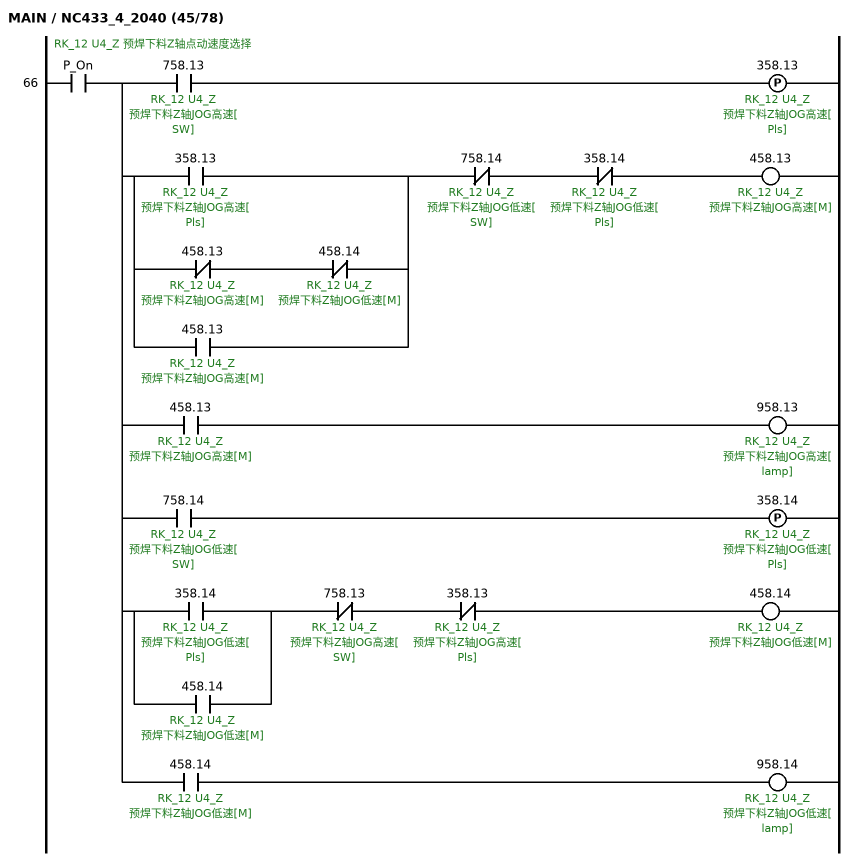
; [picture p192: MAIN / NC433_4_2040, rungs 66-66]
; rung 66: RK_12 U4_Z 预焊下料Z轴点动速度选择
LD P_On
OUT TR0
AND 758.13  ; RK_12 U4_Z 预焊下料Z轴JOG高速[SW]
DIFU(013) 358.13  ; RK_12 U4_Z 预焊下料Z轴JOG高速[Pls]
LD TR0
LD 358.13  ; RK_12 U4_Z 预焊下料Z轴JOG高速[Pls]
LDNOT 458.13  ; RK_12 U4_Z 预焊下料Z轴JOG高速[M]
ANDNOT 458.14  ; RK_12 U4_Z 预焊下料Z轴JOG低速[M]
ORLD
OR 458.13  ; RK_12 U4_Z 预焊下料Z轴JOG高速[M]
ANDLD
ANDNOT 758.14  ; RK_12 U4_Z 预焊下料Z轴JOG低速[SW]
ANDNOT 358.14  ; RK_12 U4_Z 预焊下料Z轴JOG低速[Pls]
OUT 458.13  ; RK_12 U4_Z 预焊下料Z轴JOG高速[M]
LD TR0
AND 458.13  ; RK_12 U4_Z 预焊下料Z轴JOG高速[M]
OUT 958.13  ; RK_12 U4_Z 预焊下料Z轴JOG高速[lamp]
LD TR0
AND 758.14  ; RK_12 U4_Z 预焊下料Z轴JOG低速[SW]
DIFU(013) 358.14  ; RK_12 U4_Z 预焊下料Z轴JOG低速[Pls]
LD TR0
LD 358.14  ; RK_12 U4_Z 预焊下料Z轴JOG低速[Pls]
OR 458.14  ; RK_12 U4_Z 预焊下料Z轴JOG低速[M]
ANDLD
ANDNOT 758.13  ; RK_12 U4_Z 预焊下料Z轴JOG高速[SW]
ANDNOT 358.13  ; RK_12 U4_Z 预焊下料Z轴JOG高速[Pls]
OUT 458.14  ; RK_12 U4_Z 预焊下料Z轴JOG低速[M]
LD TR0
AND 458.14  ; RK_12 U4_Z 预焊下料Z轴JOG低速[M]
OUT 958.14  ; RK_12 U4_Z 预焊下料Z轴JOG低速[lamp]

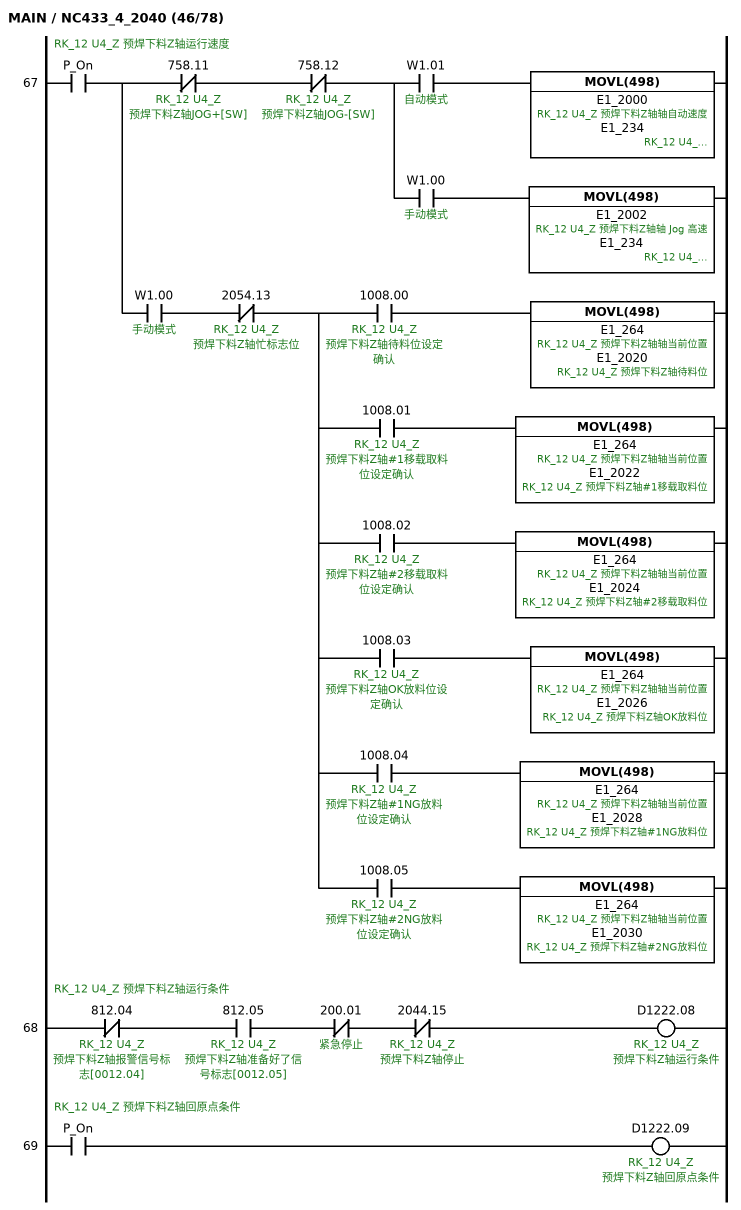
; rung 67: RK_12 U4_Z 预焊下料Z轴运行速度
LD P_On
OUT TR0
ANDNOT 758.11  ; RK_12 U4_Z 预焊下料Z轴JOG+[SW]
ANDNOT 758.12  ; RK_12 U4_Z 预焊下料Z轴JOG-[SW]
OUT TR1
AND W1.01  ; 自动模式
MOVL(498) E1_2000 E1_234  ; RK_12 U4_Z 预焊下料Z轴轴自动速度, RK_12 U4_Z 预焊下料Z轴轴直接操作速度
LD TR1
AND W1.00  ; 手动模式
MOVL(498) E1_2002 E1_234  ; RK_12 U4_Z 预焊下料Z轴轴 Jog 高速, RK_12 U4_Z 预焊下料Z轴轴直接操作速度
LD TR0
AND W1.00  ; 手动模式
ANDNOT 2054.13  ; RK_12 U4_Z 预焊下料Z轴忙标志位
OUT TR0
AND 1008.00  ; RK_12 U4_Z 预焊下料Z轴待料位设定确认
MOVL(498) E1_264 E1_2020  ; RK_12 U4_Z 预焊下料Z轴轴当前位置, RK_12 U4_Z 预焊下料Z轴待料位
LD TR0
AND 1008.01  ; RK_12 U4_Z 预焊下料Z轴#1移载取料位设定确认
MOVL(498) E1_264 E1_2022  ; RK_12 U4_Z 预焊下料Z轴轴当前位置, RK_12 U4_Z 预焊下料Z轴#1移载取料位
LD TR0
AND 1008.02  ; RK_12 U4_Z 预焊下料Z轴#2移载取料位设定确认
MOVL(498) E1_264 E1_2024  ; RK_12 U4_Z 预焊下料Z轴轴当前位置, RK_12 U4_Z 预焊下料Z轴#2移载取料位
LD TR0
AND 1008.03  ; RK_12 U4_Z 预焊下料Z轴OK放料位设定确认
MOVL(498) E1_264 E1_2026  ; RK_12 U4_Z 预焊下料Z轴轴当前位置, RK_12 U4_Z 预焊下料Z轴OK放料位
LD TR0
AND 1008.04  ; RK_12 U4_Z 预焊下料Z轴#1NG放料位设定确认
MOVL(498) E1_264 E1_2028  ; RK_12 U4_Z 预焊下料Z轴轴当前位置, RK_12 U4_Z 预焊下料Z轴#1NG放料位
LD TR0
AND 1008.05  ; RK_12 U4_Z 预焊下料Z轴#2NG放料位设定确认
MOVL(498) E1_264 E1_2030  ; RK_12 U4_Z 预焊下料Z轴轴当前位置, RK_12 U4_Z 预焊下料Z轴#2NG放料位
; rung 68: RK_12 U4_Z 预焊下料Z轴运行条件
LDNOT 812.04  ; RK_12 U4_Z 预焊下料Z轴报警信号标志[0012.04]
AND 812.05  ; RK_12 U4_Z 预焊下料Z轴准备好了信号标志[0012.05]
ANDNOT 200.01  ; 紧急停止
ANDNOT 2044.15  ; RK_12 U4_Z 预焊下料Z轴停止
OUT D1222.08  ; RK_12 U4_Z 预焊下料Z轴运行条件
; rung 69: RK_12 U4_Z 预焊下料Z轴回原点条件
LD P_On
OUT D1222.09  ; RK_12 U4_Z 预焊下料Z轴回原点条件

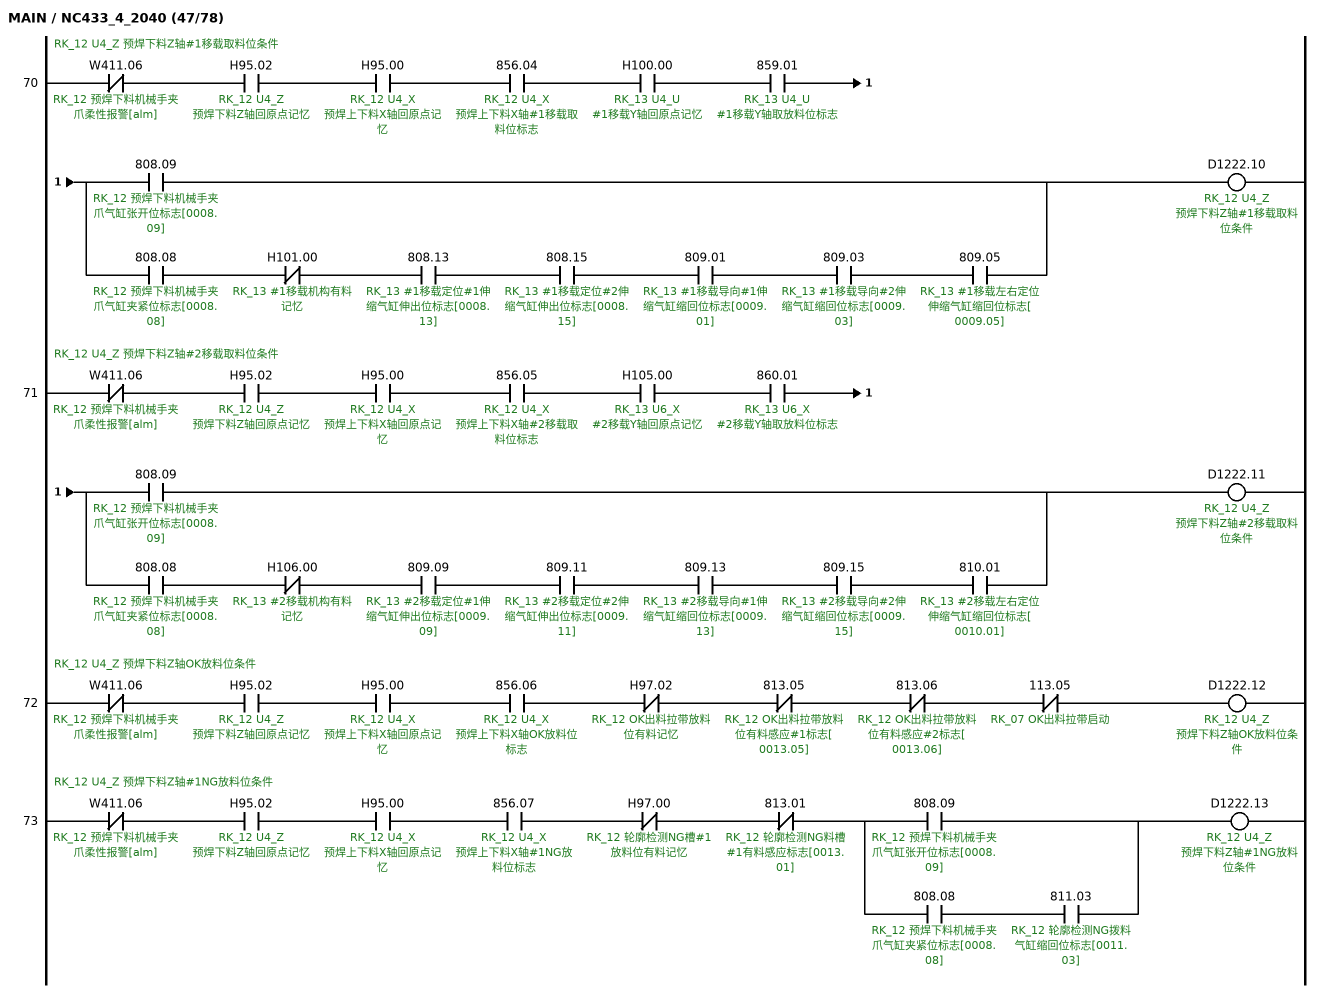
; rung 70: RK_12 U4_Z 预焊下料Z轴#1移载取料位条件
LDNOT W411.06  ; RK_12 预焊下料机械手夹爪柔性报警[alm]
AND H95.02  ; RK_12 U4_Z 预焊下料Z轴回原点记忆
AND H95.00  ; RK_12 U4_X 预焊上下料X轴回原点记忆
AND 856.04  ; RK_12 U4_X 预焊上下料X轴#1移载取料位标志
AND H100.00  ; RK_13 U4_U #1移载Y轴回原点记忆
AND 859.01  ; RK_13 U4_U #1移载Y轴取放料位标志
LD 808.09  ; RK_12 预焊下料机械手夹爪气缸张开位标志[0008.09]
LD 808.08  ; RK_12 预焊下料机械手夹爪气缸夹紧位标志[0008.08]
ANDNOT H101.00  ; RK_13 #1移载机构有料记忆
AND 808.13  ; RK_13 #1移载定位#1伸缩气缸伸出位标志[0008.13]
AND 808.15  ; RK_13 #1移载定位#2伸缩气缸伸出位标志[0008.15]
AND 809.01  ; RK_13 #1移载导向#1伸缩气缸缩回位标志[0009.01]
AND 809.03  ; RK_13 #1移载导向#2伸缩气缸缩回位标志[0009.03]
AND 809.05  ; RK_13 #1移载左右定位伸缩气缸缩回位标志[0009.05]
ORLD
ANDLD
OUT D1222.10  ; RK_12 U4_Z 预焊下料Z轴#1移载取料位条件
; rung 71: RK_12 U4_Z 预焊下料Z轴#2移载取料位条件
LDNOT W411.06  ; RK_12 预焊下料机械手夹爪柔性报警[alm]
AND H95.02  ; RK_12 U4_Z 预焊下料Z轴回原点记忆
AND H95.00  ; RK_12 U4_X 预焊上下料X轴回原点记忆
AND 856.05  ; RK_12 U4_X 预焊上下料X轴#2移载取料位标志
AND H105.00  ; RK_13 U6_X #2移载Y轴回原点记忆
AND 860.01  ; RK_13 U6_X #2移载Y轴取放料位标志
LD 808.09  ; RK_12 预焊下料机械手夹爪气缸张开位标志[0008.09]
LD 808.08  ; RK_12 预焊下料机械手夹爪气缸夹紧位标志[0008.08]
ANDNOT H106.00  ; RK_13 #2移载机构有料记忆
AND 809.09  ; RK_13 #2移载定位#1伸缩气缸伸出位标志[0009.09]
AND 809.11  ; RK_13 #2移载定位#2伸缩气缸伸出位标志[0009.11]
AND 809.13  ; RK_13 #2移载导向#1伸缩气缸缩回位标志[0009.13]
AND 809.15  ; RK_13 #2移载导向#2伸缩气缸缩回位标志[0009.15]
AND 810.01  ; RK_13 #2移载左右定位伸缩气缸缩回位标志[0010.01]
ORLD
ANDLD
OUT D1222.11  ; RK_12 U4_Z 预焊下料Z轴#2移载取料位条件
; rung 72: RK_12 U4_Z 预焊下料Z轴OK放料位条件
LDNOT W411.06  ; RK_12 预焊下料机械手夹爪柔性报警[alm]
AND H95.02  ; RK_12 U4_Z 预焊下料Z轴回原点记忆
AND H95.00  ; RK_12 U4_X 预焊上下料X轴回原点记忆
AND 856.06  ; RK_12 U4_X 预焊上下料X轴OK放料位标志
ANDNOT H97.02  ; RK_12 OK出料拉带放料位有料记忆  // RK_12 OK出料拉带放料位有料记忆+OK出料拉带放料位有料感应标志+拉带电机未启动标志！！
ANDNOT 813.05  ; RK_12 OK出料拉带放料位有料感应#1标志[0013.05]
ANDNOT 813.06  ; RK_12 OK出料拉带放料位有料感应#2标志[0013.06]
ANDNOT 113.05  ; RK_07 OK出料拉带启动
OUT D1222.12  ; RK_12 U4_Z 预焊下料Z轴OK放料位条件
; rung 73: RK_12 U4_Z 预焊下料Z轴#1NG放料位条件
LDNOT W411.06  ; RK_12 预焊下料机械手夹爪柔性报警[alm]
AND H95.02  ; RK_12 U4_Z 预焊下料Z轴回原点记忆
AND H95.00  ; RK_12 U4_X 预焊上下料X轴回原点记忆
AND 856.07  ; RK_12 U4_X 预焊上下料X轴#1NG放料位标志
ANDNOT H97.00  ; RK_12 轮廓检测NG槽#1放料位有料记忆
ANDNOT 813.01  ; RK_12 轮廓检测NG料槽#1有料感应标志[0013.01]
LD 808.09  ; RK_12 预焊下料机械手夹爪气缸张开位标志[0008.09]
LD 808.08  ; RK_12 预焊下料机械手夹爪气缸夹紧位标志[0008.08]
AND 811.03  ; RK_12 轮廓检测NG拨料气缸缩回位标志[0011.03]
ORLD
ANDLD
OUT D1222.13  ; RK_12 U4_Z 预焊下料Z轴#1NG放料位条件

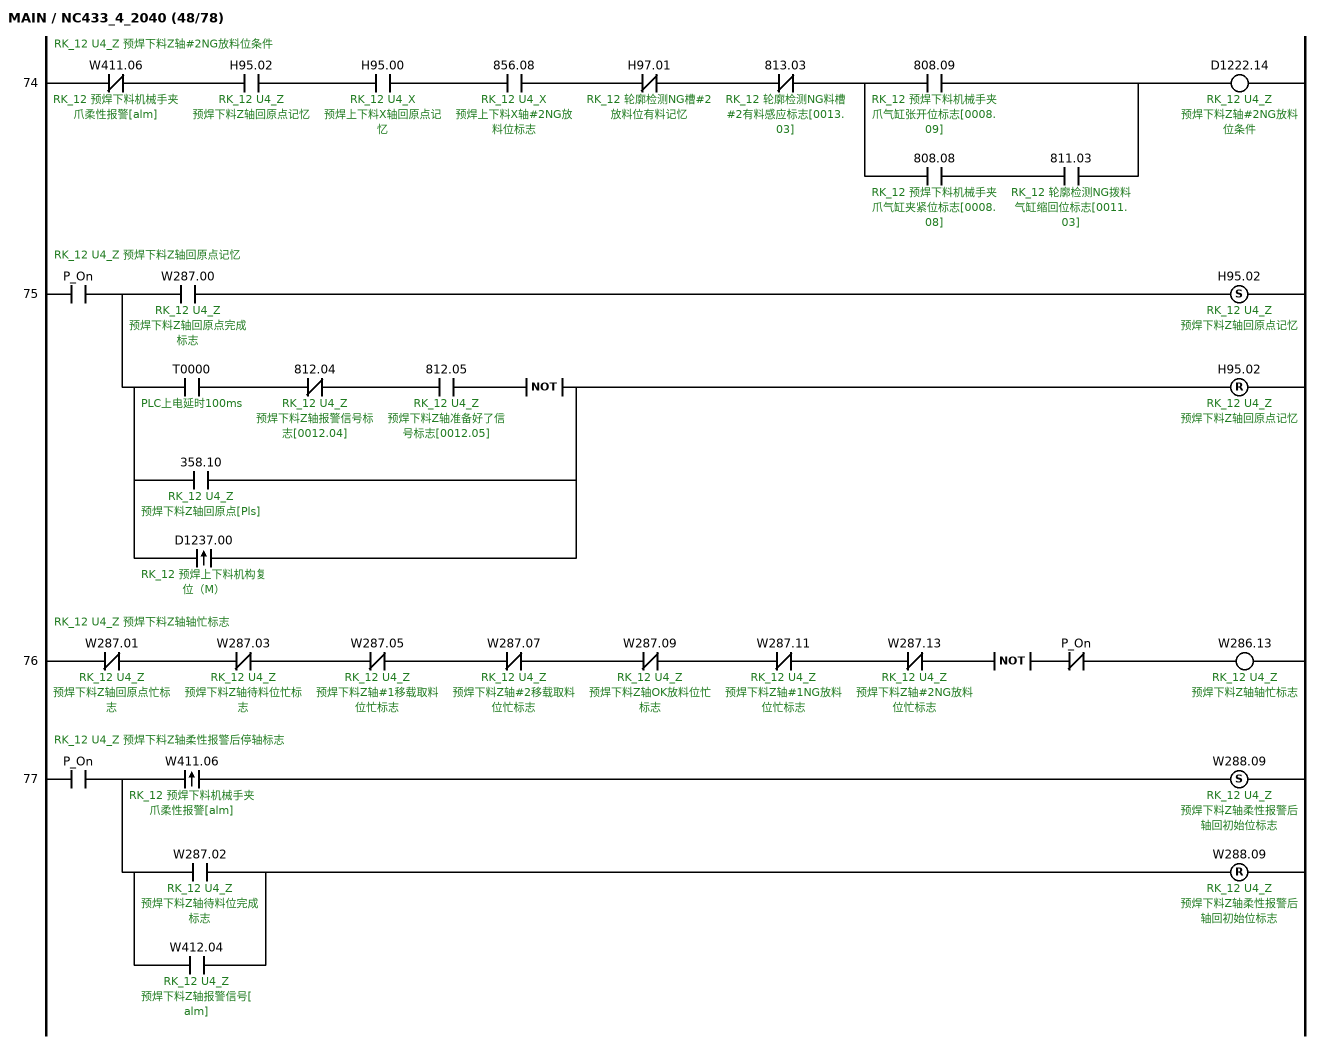
; rung 74: RK_12 U4_Z 预焊下料Z轴#2NG放料位条件
LDNOT W411.06  ; RK_12 预焊下料机械手夹爪柔性报警[alm]
AND H95.02  ; RK_12 U4_Z 预焊下料Z轴回原点记忆
AND H95.00  ; RK_12 U4_X 预焊上下料X轴回原点记忆
AND 856.08  ; RK_12 U4_X 预焊上下料X轴#2NG放料位标志
ANDNOT H97.01  ; RK_12 轮廓检测NG槽#2放料位有料记忆
ANDNOT 813.03  ; RK_12 轮廓检测NG料槽#2有料感应标志[0013.03]
LD 808.09  ; RK_12 预焊下料机械手夹爪气缸张开位标志[0008.09]
LD 808.08  ; RK_12 预焊下料机械手夹爪气缸夹紧位标志[0008.08]
AND 811.03  ; RK_12 轮廓检测NG拨料气缸缩回位标志[0011.03]
ORLD
ANDLD
OUT D1222.14  ; RK_12 U4_Z 预焊下料Z轴#2NG放料位条件
; rung 75: RK_12 U4_Z 预焊下料Z轴回原点记忆
LD P_On
OUT TR0
AND W287.00  ; RK_12 U4_Z 预焊下料Z轴回原点完成标志
SET H95.02  ; RK_12 U4_Z 预焊下料Z轴回原点记忆
LD TR0
LD T0000  ; PLC上电延时100ms
ANDNOT 812.04  ; RK_12 U4_Z 预焊下料Z轴报警信号标志[0012.04]
AND 812.05  ; RK_12 U4_Z 预焊下料Z轴准备好了信号标志[0012.05]
NOT(520)
OR 358.10  ; RK_12 U4_Z 预焊下料Z轴回原点[Pls]
@OR D1237.00  ; RK_12 预焊上下料机构复位（M）
ANDLD
RSET H95.02  ; RK_12 U4_Z 预焊下料Z轴回原点记忆
; rung 76: RK_12 U4_Z 预焊下料Z轴轴忙标志
LDNOT W287.01  ; RK_12 U4_Z 预焊下料Z轴回原点忙标志
ANDNOT W287.03  ; RK_12 U4_Z 预焊下料Z轴待料位忙标志
ANDNOT W287.05  ; RK_12 U4_Z 预焊下料Z轴#1移载取料位忙标志
ANDNOT W287.07  ; RK_12 U4_Z 预焊下料Z轴#2移载取料位忙标志
ANDNOT W287.09  ; RK_12 U4_Z 预焊下料Z轴OK放料位忙标志
ANDNOT W287.11  ; RK_12 U4_Z 预焊下料Z轴#1NG放料位忙标志
ANDNOT W287.13  ; RK_12 U4_Z 预焊下料Z轴#2NG放料位忙标志
NOT(520)
ANDNOT P_On
OUT W286.13  ; RK_12 U4_Z 预焊下料Z轴轴忙标志
; rung 77: RK_12 U4_Z 预焊下料Z轴柔性报警后停轴标志
LD P_On
OUT TR0
@AND W411.06  ; RK_12 预焊下料机械手夹爪柔性报警[alm]
SET W288.09  ; RK_12 U4_Z 预焊下料Z轴柔性报警后轴回初始位标志
LD TR0
LD W287.02  ; RK_12 U4_Z 预焊下料Z轴待料位完成标志
OR W412.04  ; RK_12 U4_Z 预焊下料Z轴报警信号[alm]
ANDLD
RSET W288.09  ; RK_12 U4_Z 预焊下料Z轴柔性报警后轴回初始位标志

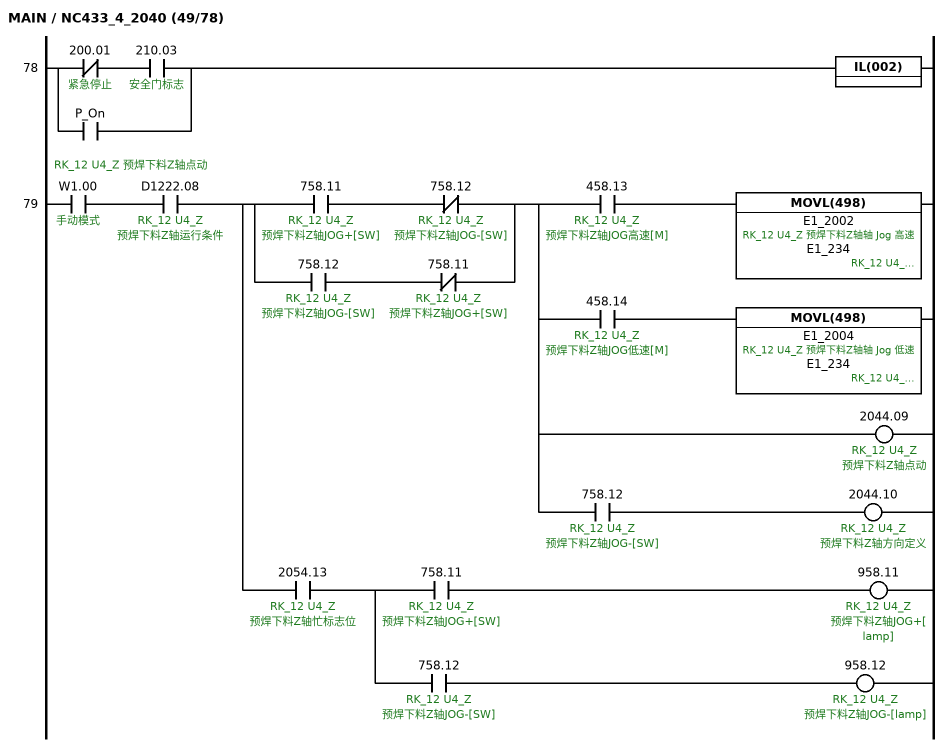
; rung 78
LDNOT 200.01  ; 紧急停止
AND 210.03  ; 安全门标志
OR P_On
IL(002)
; rung 79: RK_12 U4_Z 预焊下料Z轴点动
LD W1.00  ; 手动模式
AND D1222.08  ; RK_12 U4_Z 预焊下料Z轴运行条件
OUT TR0
LD 758.11  ; RK_12 U4_Z 预焊下料Z轴JOG+[SW]
ANDNOT 758.12  ; RK_12 U4_Z 预焊下料Z轴JOG-[SW]
LD 758.12  ; RK_12 U4_Z 预焊下料Z轴JOG-[SW]
ANDNOT 758.11  ; RK_12 U4_Z 预焊下料Z轴JOG+[SW]
ORLD
ANDLD
OUT TR1
AND 458.13  ; RK_12 U4_Z 预焊下料Z轴JOG高速[M]
MOVL(498) E1_2002 E1_234  ; RK_12 U4_Z 预焊下料Z轴轴 Jog 高速, RK_12 U4_Z 预焊下料Z轴轴直接操作速度
LD TR1
AND 458.14  ; RK_12 U4_Z 预焊下料Z轴JOG低速[M]
MOVL(498) E1_2004 E1_234  ; RK_12 U4_Z 预焊下料Z轴轴 Jog 低速, RK_12 U4_Z 预焊下料Z轴轴直接操作速度
LD TR1
OUT 2044.09  ; RK_12 U4_Z 预焊下料Z轴点动
AND 758.12  ; RK_12 U4_Z 预焊下料Z轴JOG-[SW]
OUT 2044.10  ; RK_12 U4_Z 预焊下料Z轴方向定义
LD TR0
AND 2054.13  ; RK_12 U4_Z 预焊下料Z轴忙标志位
OUT TR0
AND 758.11  ; RK_12 U4_Z 预焊下料Z轴JOG+[SW]
OUT 958.11  ; RK_12 U4_Z 预焊下料Z轴JOG+[lamp]
LD TR0
AND 758.12  ; RK_12 U4_Z 预焊下料Z轴JOG-[SW]
OUT 958.12  ; RK_12 U4_Z 预焊下料Z轴JOG-[lamp]

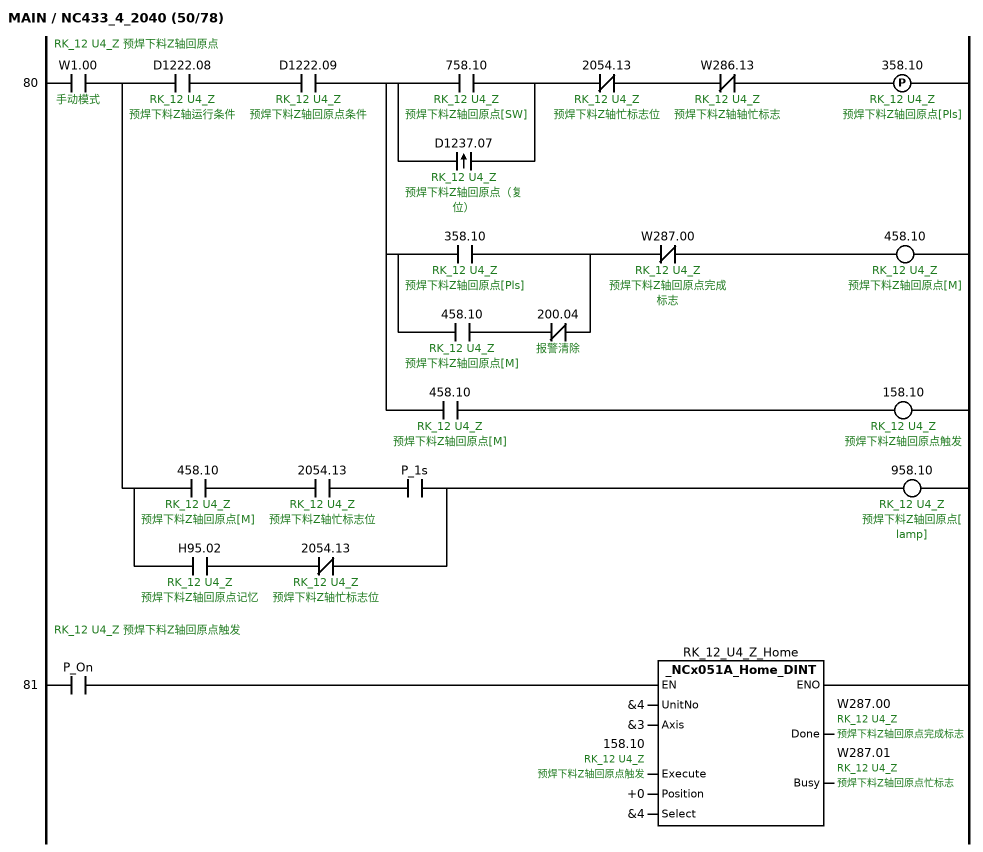
; rung 80: RK_12 U4_Z 预焊下料Z轴回原点
LD W1.00  ; 手动模式
OUT TR0
AND D1222.08  ; RK_12 U4_Z 预焊下料Z轴运行条件
AND D1222.09  ; RK_12 U4_Z 预焊下料Z轴回原点条件
OUT TR1
LD 758.10  ; RK_12 U4_Z 预焊下料Z轴回原点[SW]
@OR D1237.07  ; RK_12 U4_Z 预焊下料Z轴回原点（复位）
ANDLD
ANDNOT 2054.13  ; RK_12 U4_Z 预焊下料Z轴忙标志位
ANDNOT W286.13  ; RK_12 U4_Z 预焊下料Z轴轴忙标志
DIFU(013) 358.10  ; RK_12 U4_Z 预焊下料Z轴回原点[Pls]
LD TR1
LD 358.10  ; RK_12 U4_Z 预焊下料Z轴回原点[Pls]
LD 458.10  ; RK_12 U4_Z 预焊下料Z轴回原点[M]
ANDNOT 200.04  ; 报警清除
ORLD
ANDLD
ANDNOT W287.00  ; RK_12 U4_Z 预焊下料Z轴回原点完成标志
OUT 458.10  ; RK_12 U4_Z 预焊下料Z轴回原点[M]
LD TR1
AND 458.10  ; RK_12 U4_Z 预焊下料Z轴回原点[M]
OUT 158.10  ; RK_12 U4_Z 预焊下料Z轴回原点触发
LD TR0
LD 458.10  ; RK_12 U4_Z 预焊下料Z轴回原点[M]
AND 2054.13  ; RK_12 U4_Z 预焊下料Z轴忙标志位
AND P_1s
LD H95.02  ; RK_12 U4_Z 预焊下料Z轴回原点记忆
ANDNOT 2054.13  ; RK_12 U4_Z 预焊下料Z轴忙标志位
ORLD
ANDLD
OUT 958.10  ; RK_12 U4_Z 预焊下料Z轴回原点[lamp]
; rung 81: RK_12 U4_Z 预焊下料Z轴回原点触发
LD P_On
CALL RK_12_U4_Z_Home : _NCx051A_Home_DINT (UnitNo := &4, Axis := &3, Execute := 158.10, Position := +0, Select := &4, Done => W287.00, Busy => W287.01)  ; RK_12 U4_Z 预焊下料Z轴回原点触发, RK_12 U4_Z 预焊下料Z轴回原点完成标志, RK_12 U4_Z 预焊下料Z轴回原点忙标志

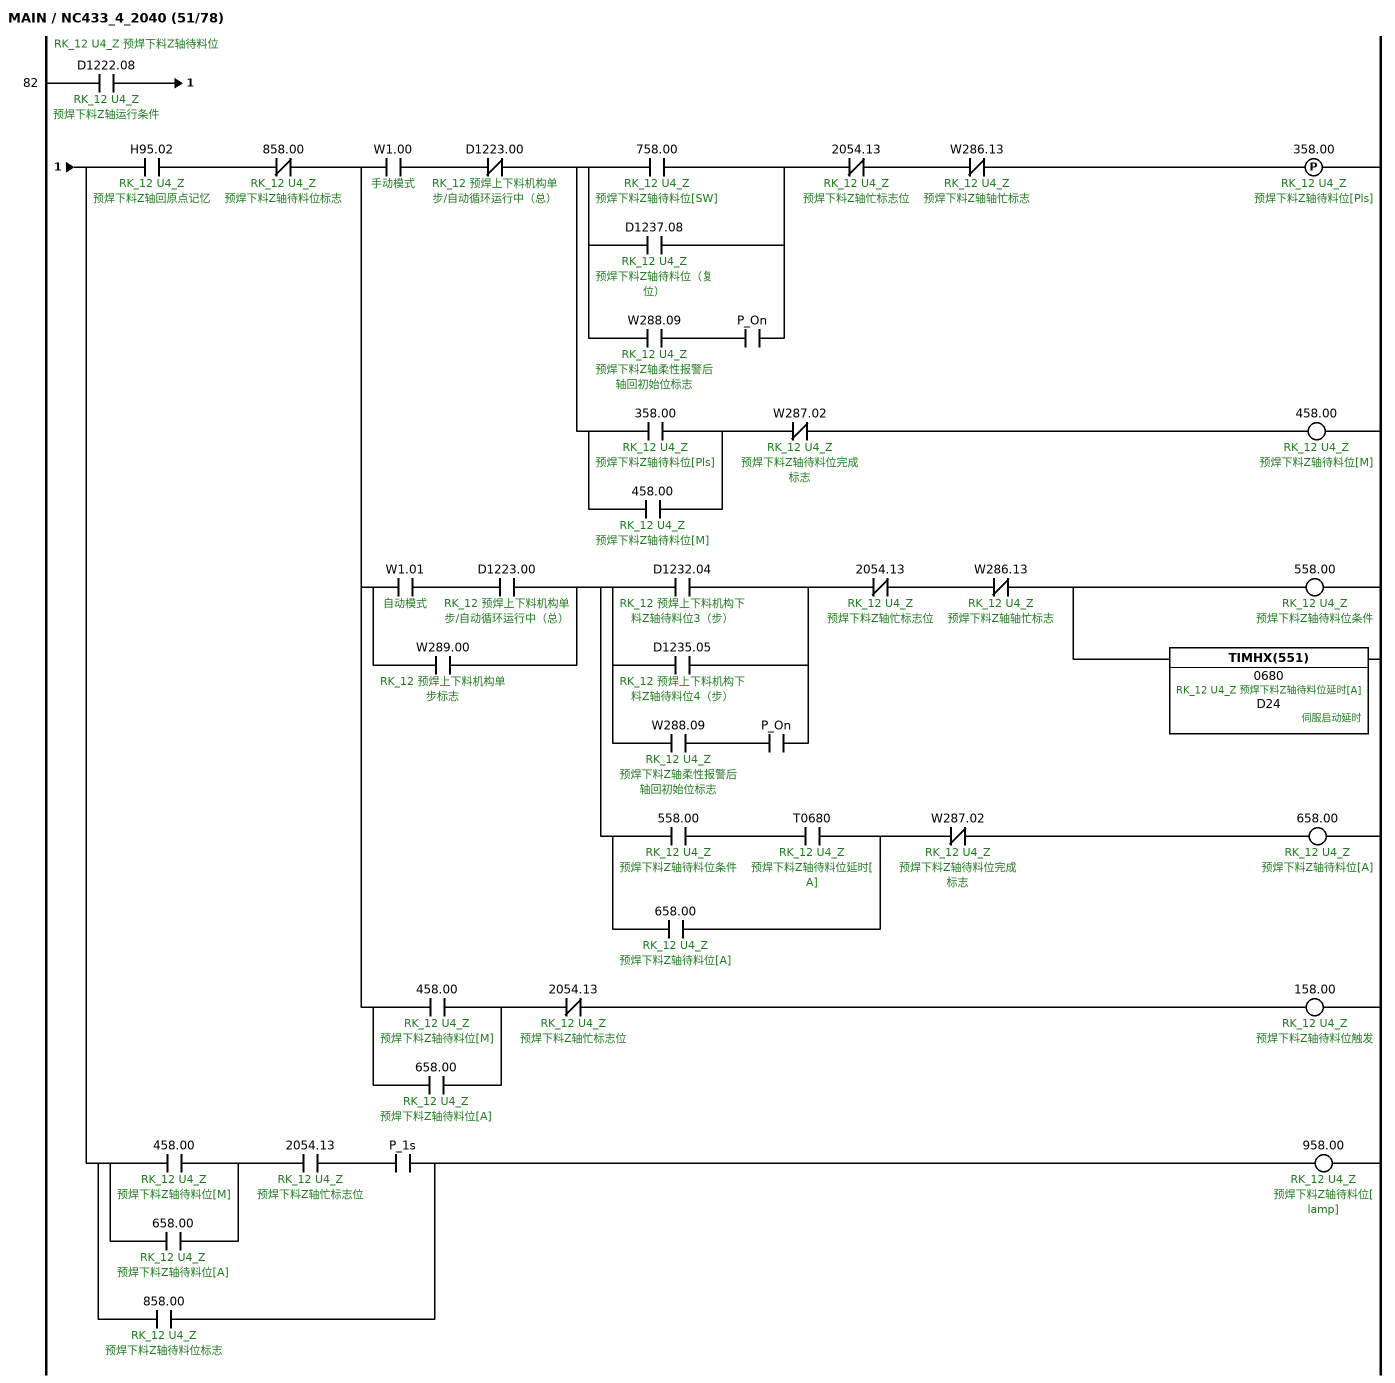
; rung 82: RK_12 U4_Z 预焊下料Z轴待料位
LD D1222.08  ; RK_12 U4_Z 预焊下料Z轴运行条件
OUT TR0
AND H95.02  ; RK_12 U4_Z 预焊下料Z轴回原点记忆
ANDNOT 858.00  ; RK_12 U4_Z 预焊下料Z轴待料位标志
OUT TR1
AND W1.00  ; 手动模式
ANDNOT D1223.00  ; RK_12 预焊上下料机构单步/自动循环运行中（总）
OUT TR2
LD 758.00  ; RK_12 U4_Z 预焊下料Z轴待料位[SW]
OR D1237.08  ; RK_12 U4_Z 预焊下料Z轴待料位（复位）
LD W288.09  ; RK_12 U4_Z 预焊下料Z轴柔性报警后轴回初始位标志
AND P_On
ORLD
ANDLD
ANDNOT 2054.13  ; RK_12 U4_Z 预焊下料Z轴忙标志位
ANDNOT W286.13  ; RK_12 U4_Z 预焊下料Z轴轴忙标志
DIFU(013) 358.00  ; RK_12 U4_Z 预焊下料Z轴待料位[Pls]
LD TR2
LD 358.00  ; RK_12 U4_Z 预焊下料Z轴待料位[Pls]
OR 458.00  ; RK_12 U4_Z 预焊下料Z轴待料位[M]
ANDLD
ANDNOT W287.02  ; RK_12 U4_Z 预焊下料Z轴待料位完成标志
OUT 458.00  ; RK_12 U4_Z 预焊下料Z轴待料位[M]
LD TR1
LD W1.01  ; 自动模式
AND D1223.00  ; RK_12 预焊上下料机构单步/自动循环运行中（总）
OR W289.00  ; RK_12 预焊上下料机构单步标志
ANDLD
OUT TR2
LD D1232.04  ; RK_12 预焊上下料机构下料Z轴待料位3（步）
OR D1235.05  ; RK_12 预焊上下料机构下料Z轴待料位4（步）
LD W288.09  ; RK_12 U4_Z 预焊下料Z轴柔性报警后轴回初始位标志
AND P_On
ORLD
ANDLD
ANDNOT 2054.13  ; RK_12 U4_Z 预焊下料Z轴忙标志位
ANDNOT W286.13  ; RK_12 U4_Z 预焊下料Z轴轴忙标志
OUT 558.00  ; RK_12 U4_Z 预焊下料Z轴待料位条件
TIMHX(551) 0680 D24  ; 伺服启动延时, RK_12 U4_Z 预焊下料Z轴待料位延时[A]
LD TR2
LD 558.00  ; RK_12 U4_Z 预焊下料Z轴待料位条件
AND T0680  ; RK_12 U4_Z 预焊下料Z轴待料位延时[A]
OR 658.00  ; RK_12 U4_Z 预焊下料Z轴待料位[A]
ANDLD
ANDNOT W287.02  ; RK_12 U4_Z 预焊下料Z轴待料位完成标志
OUT 658.00  ; RK_12 U4_Z 预焊下料Z轴待料位[A]
LD TR1
LD 458.00  ; RK_12 U4_Z 预焊下料Z轴待料位[M]
OR 658.00  ; RK_12 U4_Z 预焊下料Z轴待料位[A]
ANDLD
ANDNOT 2054.13  ; RK_12 U4_Z 预焊下料Z轴忙标志位
OUT 158.00  ; RK_12 U4_Z 预焊下料Z轴待料位触发
LD TR0
LD 458.00  ; RK_12 U4_Z 预焊下料Z轴待料位[M]
OR 658.00  ; RK_12 U4_Z 预焊下料Z轴待料位[A]
AND 2054.13  ; RK_12 U4_Z 预焊下料Z轴忙标志位
AND P_1s
OR 858.00  ; RK_12 U4_Z 预焊下料Z轴待料位标志
ANDLD
OUT 958.00  ; RK_12 U4_Z 预焊下料Z轴待料位[lamp]

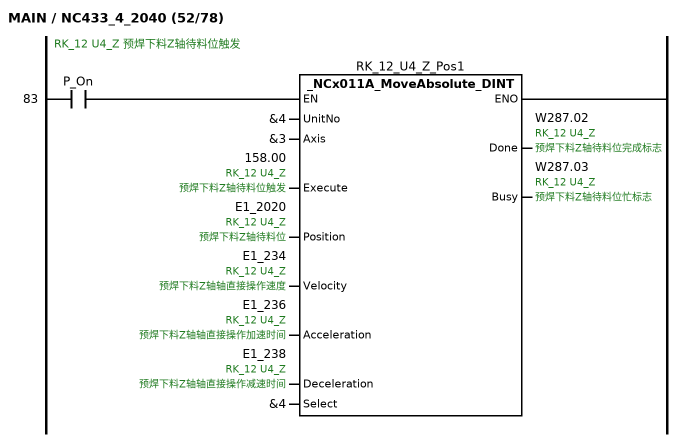
; rung 83: RK_12 U4_Z 预焊下料Z轴待料位触发
LD P_On
CALL RK_12_U4_Z_Pos1 : _NCx011A_MoveAbsolute_DINT (UnitNo := &4, Axis := &3, Execute := 158.00, Position := E1_2020, Velocity := E1_234, Acceleration := E1_236, Deceleration := E1_238, Select := &4, Done => W287.02, Busy => W287.03)  ; RK_12 U4_Z 预焊下料Z轴待料位触发, RK_12 U4_Z 预焊下料Z轴待料位, RK_12 U4_Z 预焊下料Z轴轴直接操作速度, RK_12 U4_Z 预焊下料Z轴轴直接操作加速时间, RK_12 U4_Z 预焊下料Z轴轴直接操作减速时间, RK_12 U4_Z 预焊下料Z轴待料位完成标志, RK_12 U4_Z 预焊下料Z轴待料位忙标志

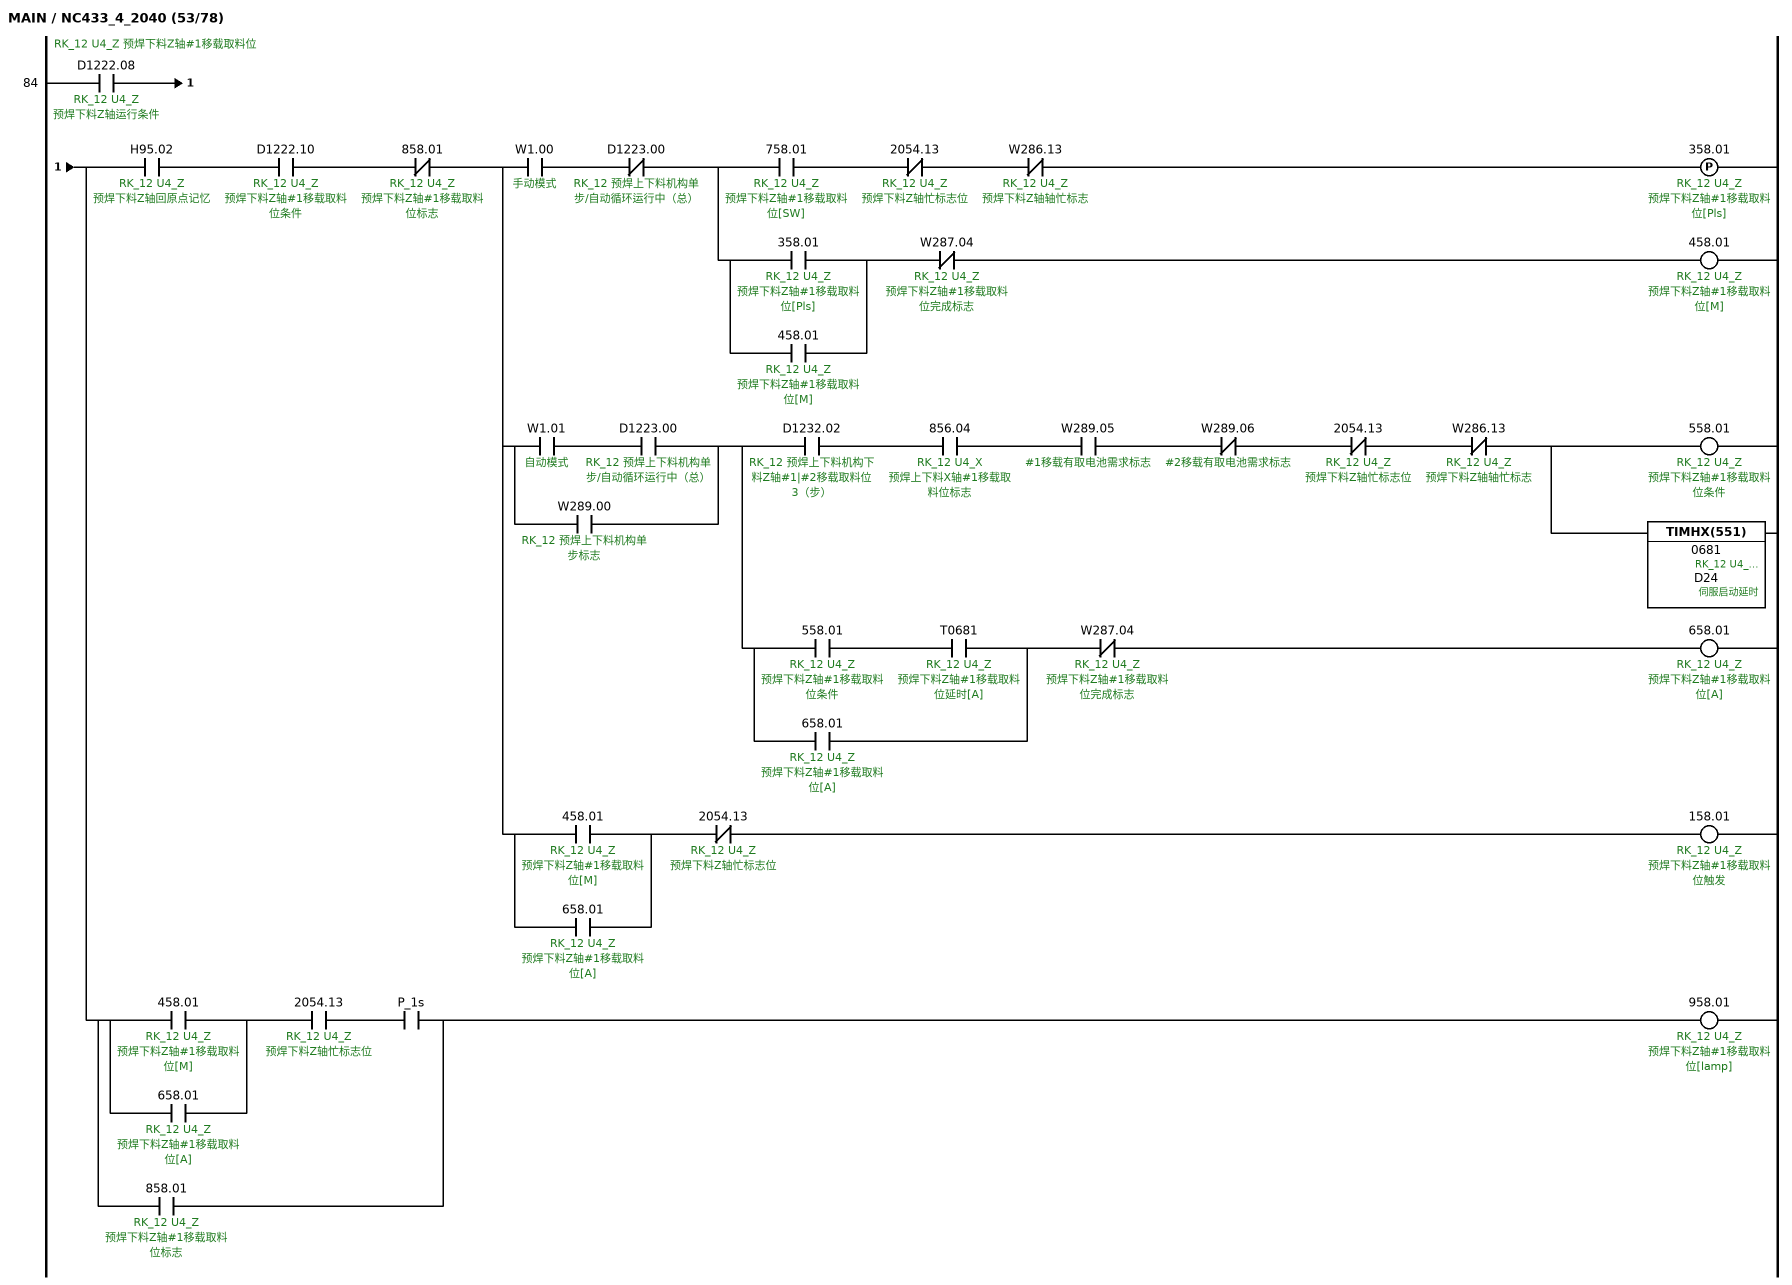
; rung 84: RK_12 U4_Z 预焊下料Z轴#1移载取料位
LD D1222.08  ; RK_12 U4_Z 预焊下料Z轴运行条件
OUT TR0
AND H95.02  ; RK_12 U4_Z 预焊下料Z轴回原点记忆
AND D1222.10  ; RK_12 U4_Z 预焊下料Z轴#1移载取料位条件
ANDNOT 858.01  ; RK_12 U4_Z 预焊下料Z轴#1移载取料位标志
OUT TR1
AND W1.00  ; 手动模式
ANDNOT D1223.00  ; RK_12 预焊上下料机构单步/自动循环运行中（总）
OUT TR2
AND 758.01  ; RK_12 U4_Z 预焊下料Z轴#1移载取料位[SW]
ANDNOT 2054.13  ; RK_12 U4_Z 预焊下料Z轴忙标志位
ANDNOT W286.13  ; RK_12 U4_Z 预焊下料Z轴轴忙标志
DIFU(013) 358.01  ; RK_12 U4_Z 预焊下料Z轴#1移载取料位[Pls]
LD TR2
LD 358.01  ; RK_12 U4_Z 预焊下料Z轴#1移载取料位[Pls]
OR 458.01  ; RK_12 U4_Z 预焊下料Z轴#1移载取料位[M]
ANDLD
ANDNOT W287.04  ; RK_12 U4_Z 预焊下料Z轴#1移载取料位完成标志
OUT 458.01  ; RK_12 U4_Z 预焊下料Z轴#1移载取料位[M]
LD TR1
LD W1.01  ; 自动模式
AND D1223.00  ; RK_12 预焊上下料机构单步/自动循环运行中（总）
OR W289.00  ; RK_12 预焊上下料机构单步标志
ANDLD
OUT TR2
AND D1232.02  ; RK_12 预焊上下料机构下料Z轴#1|#2移载取料位3（步）
AND 856.04  ; RK_12 U4_X 预焊上下料X轴#1移载取料位标志
AND W289.05  ; #1移载有取电池需求标志
ANDNOT W289.06  ; #2移载有取电池需求标志
ANDNOT 2054.13  ; RK_12 U4_Z 预焊下料Z轴忙标志位
ANDNOT W286.13  ; RK_12 U4_Z 预焊下料Z轴轴忙标志
OUT 558.01  ; RK_12 U4_Z 预焊下料Z轴#1移载取料位条件
TIMHX(551) 0681 D24  ; 伺服启动延时, RK_12 U4_Z 预焊下料Z轴#1移载取料位延时[A]
LD TR2
LD 558.01  ; RK_12 U4_Z 预焊下料Z轴#1移载取料位条件
AND T0681  ; RK_12 U4_Z 预焊下料Z轴#1移载取料位延时[A]
OR 658.01  ; RK_12 U4_Z 预焊下料Z轴#1移载取料位[A]
ANDLD
ANDNOT W287.04  ; RK_12 U4_Z 预焊下料Z轴#1移载取料位完成标志
OUT 658.01  ; RK_12 U4_Z 预焊下料Z轴#1移载取料位[A]
LD TR1
LD 458.01  ; RK_12 U4_Z 预焊下料Z轴#1移载取料位[M]
OR 658.01  ; RK_12 U4_Z 预焊下料Z轴#1移载取料位[A]
ANDLD
ANDNOT 2054.13  ; RK_12 U4_Z 预焊下料Z轴忙标志位
OUT 158.01  ; RK_12 U4_Z 预焊下料Z轴#1移载取料位触发
LD TR0
LD 458.01  ; RK_12 U4_Z 预焊下料Z轴#1移载取料位[M]
OR 658.01  ; RK_12 U4_Z 预焊下料Z轴#1移载取料位[A]
AND 2054.13  ; RK_12 U4_Z 预焊下料Z轴忙标志位
AND P_1s
OR 858.01  ; RK_12 U4_Z 预焊下料Z轴#1移载取料位标志
ANDLD
OUT 958.01  ; RK_12 U4_Z 预焊下料Z轴#1移载取料位[lamp]

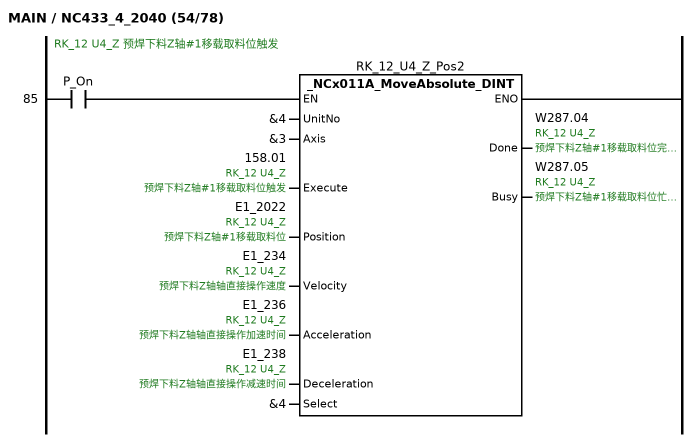
; rung 85: RK_12 U4_Z 预焊下料Z轴#1移载取料位触发
LD P_On
CALL RK_12_U4_Z_Pos2 : _NCx011A_MoveAbsolute_DINT (UnitNo := &4, Axis := &3, Execute := 158.01, Position := E1_2022, Velocity := E1_234, Acceleration := E1_236, Deceleration := E1_238, Select := &4, Done => W287.04, Busy => W287.05)  ; RK_12 U4_Z 预焊下料Z轴#1移载取料位触发, RK_12 U4_Z 预焊下料Z轴#1移载取料位, RK_12 U4_Z 预焊下料Z轴轴直接操作速度, RK_12 U4_Z 预焊下料Z轴轴直接操作加速时间, RK_12 U4_Z 预焊下料Z轴轴直接操作减速时间, RK_12 U4_Z 预焊下料Z轴#1移载取料位完成标志, RK_12 U4_Z 预焊下料Z轴#1移载取料位忙标志

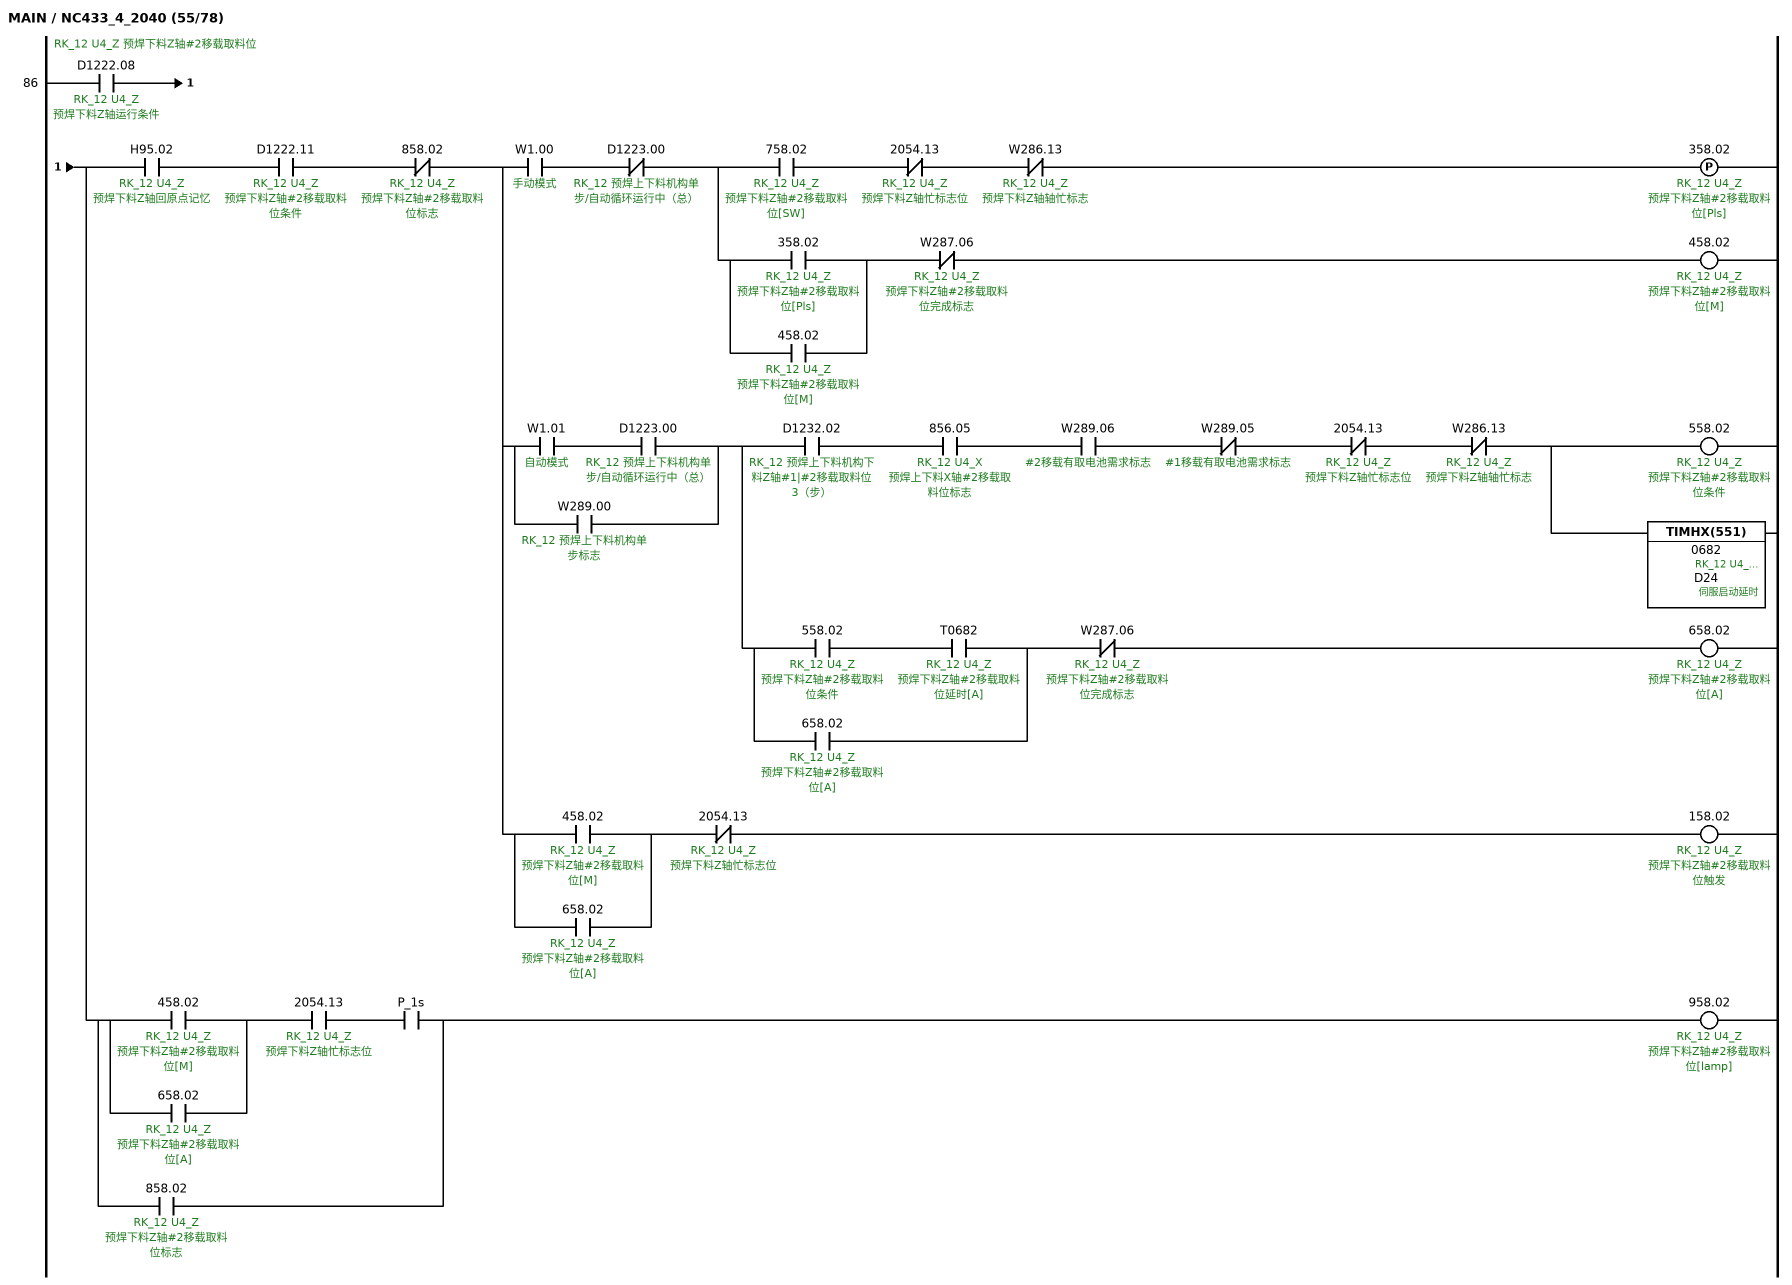
; rung 86: RK_12 U4_Z 预焊下料Z轴#2移载取料位
LD D1222.08  ; RK_12 U4_Z 预焊下料Z轴运行条件
OUT TR0
AND H95.02  ; RK_12 U4_Z 预焊下料Z轴回原点记忆
AND D1222.11  ; RK_12 U4_Z 预焊下料Z轴#2移载取料位条件
ANDNOT 858.02  ; RK_12 U4_Z 预焊下料Z轴#2移载取料位标志
OUT TR1
AND W1.00  ; 手动模式
ANDNOT D1223.00  ; RK_12 预焊上下料机构单步/自动循环运行中（总）
OUT TR2
AND 758.02  ; RK_12 U4_Z 预焊下料Z轴#2移载取料位[SW]
ANDNOT 2054.13  ; RK_12 U4_Z 预焊下料Z轴忙标志位
ANDNOT W286.13  ; RK_12 U4_Z 预焊下料Z轴轴忙标志
DIFU(013) 358.02  ; RK_12 U4_Z 预焊下料Z轴#2移载取料位[Pls]
LD TR2
LD 358.02  ; RK_12 U4_Z 预焊下料Z轴#2移载取料位[Pls]
OR 458.02  ; RK_12 U4_Z 预焊下料Z轴#2移载取料位[M]
ANDLD
ANDNOT W287.06  ; RK_12 U4_Z 预焊下料Z轴#2移载取料位完成标志
OUT 458.02  ; RK_12 U4_Z 预焊下料Z轴#2移载取料位[M]
LD TR1
LD W1.01  ; 自动模式
AND D1223.00  ; RK_12 预焊上下料机构单步/自动循环运行中（总）
OR W289.00  ; RK_12 预焊上下料机构单步标志
ANDLD
OUT TR2
AND D1232.02  ; RK_12 预焊上下料机构下料Z轴#1|#2移载取料位3（步）
AND 856.05  ; RK_12 U4_X 预焊上下料X轴#2移载取料位标志
AND W289.06  ; #2移载有取电池需求标志
ANDNOT W289.05  ; #1移载有取电池需求标志
ANDNOT 2054.13  ; RK_12 U4_Z 预焊下料Z轴忙标志位
ANDNOT W286.13  ; RK_12 U4_Z 预焊下料Z轴轴忙标志
OUT 558.02  ; RK_12 U4_Z 预焊下料Z轴#2移载取料位条件
TIMHX(551) 0682 D24  ; 伺服启动延时, RK_12 U4_Z 预焊下料Z轴#2移载取料位延时[A]
LD TR2
LD 558.02  ; RK_12 U4_Z 预焊下料Z轴#2移载取料位条件
AND T0682  ; RK_12 U4_Z 预焊下料Z轴#2移载取料位延时[A]
OR 658.02  ; RK_12 U4_Z 预焊下料Z轴#2移载取料位[A]
ANDLD
ANDNOT W287.06  ; RK_12 U4_Z 预焊下料Z轴#2移载取料位完成标志
OUT 658.02  ; RK_12 U4_Z 预焊下料Z轴#2移载取料位[A]
LD TR1
LD 458.02  ; RK_12 U4_Z 预焊下料Z轴#2移载取料位[M]
OR 658.02  ; RK_12 U4_Z 预焊下料Z轴#2移载取料位[A]
ANDLD
ANDNOT 2054.13  ; RK_12 U4_Z 预焊下料Z轴忙标志位
OUT 158.02  ; RK_12 U4_Z 预焊下料Z轴#2移载取料位触发
LD TR0
LD 458.02  ; RK_12 U4_Z 预焊下料Z轴#2移载取料位[M]
OR 658.02  ; RK_12 U4_Z 预焊下料Z轴#2移载取料位[A]
AND 2054.13  ; RK_12 U4_Z 预焊下料Z轴忙标志位
AND P_1s
OR 858.02  ; RK_12 U4_Z 预焊下料Z轴#2移载取料位标志
ANDLD
OUT 958.02  ; RK_12 U4_Z 预焊下料Z轴#2移载取料位[lamp]

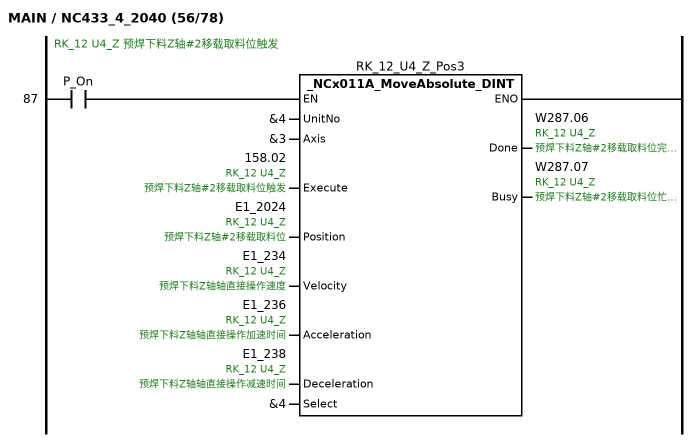
; rung 87: RK_12 U4_Z 预焊下料Z轴#2移载取料位触发
LD P_On
CALL RK_12_U4_Z_Pos3 : _NCx011A_MoveAbsolute_DINT (UnitNo := &4, Axis := &3, Execute := 158.02, Position := E1_2024, Velocity := E1_234, Acceleration := E1_236, Deceleration := E1_238, Select := &4, Done => W287.06, Busy => W287.07)  ; RK_12 U4_Z 预焊下料Z轴#2移载取料位触发, RK_12 U4_Z 预焊下料Z轴#2移载取料位, RK_12 U4_Z 预焊下料Z轴轴直接操作速度, RK_12 U4_Z 预焊下料Z轴轴直接操作加速时间, RK_12 U4_Z 预焊下料Z轴轴直接操作减速时间, RK_12 U4_Z 预焊下料Z轴#2移载取料位完成标志, RK_12 U4_Z 预焊下料Z轴#2移载取料位忙标志

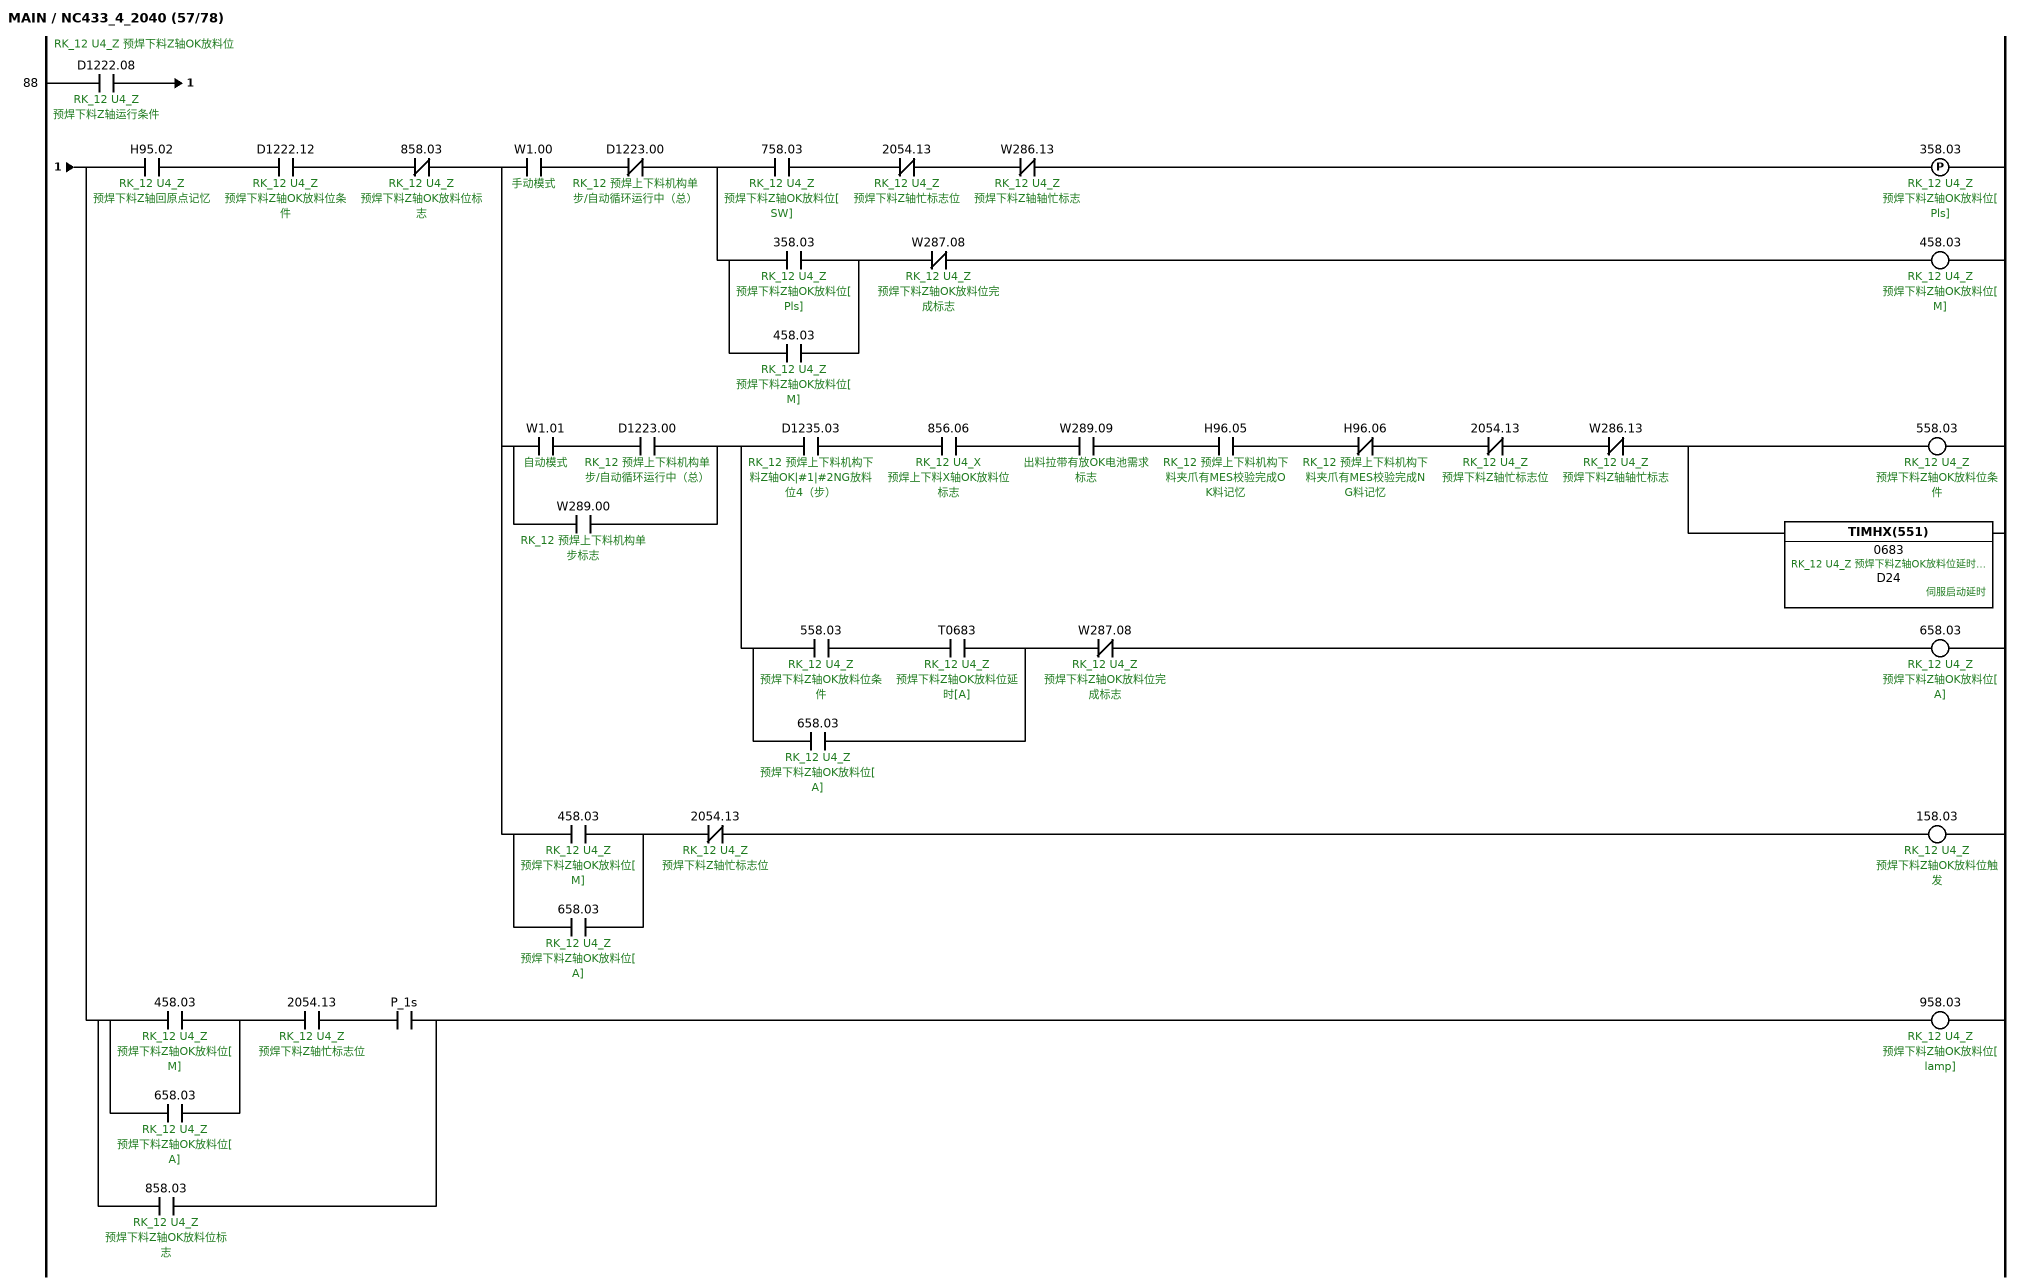
; rung 88: RK_12 U4_Z 预焊下料Z轴OK放料位
LD D1222.08  ; RK_12 U4_Z 预焊下料Z轴运行条件
OUT TR0
AND H95.02  ; RK_12 U4_Z 预焊下料Z轴回原点记忆
AND D1222.12  ; RK_12 U4_Z 预焊下料Z轴OK放料位条件
ANDNOT 858.03  ; RK_12 U4_Z 预焊下料Z轴OK放料位标志
OUT TR1
AND W1.00  ; 手动模式
ANDNOT D1223.00  ; RK_12 预焊上下料机构单步/自动循环运行中（总）
OUT TR2
AND 758.03  ; RK_12 U4_Z 预焊下料Z轴OK放料位[SW]
ANDNOT 2054.13  ; RK_12 U4_Z 预焊下料Z轴忙标志位
ANDNOT W286.13  ; RK_12 U4_Z 预焊下料Z轴轴忙标志
DIFU(013) 358.03  ; RK_12 U4_Z 预焊下料Z轴OK放料位[Pls]
LD TR2
LD 358.03  ; RK_12 U4_Z 预焊下料Z轴OK放料位[Pls]
OR 458.03  ; RK_12 U4_Z 预焊下料Z轴OK放料位[M]
ANDLD
ANDNOT W287.08  ; RK_12 U4_Z 预焊下料Z轴OK放料位完成标志
OUT 458.03  ; RK_12 U4_Z 预焊下料Z轴OK放料位[M]
LD TR1
LD W1.01  ; 自动模式
AND D1223.00  ; RK_12 预焊上下料机构单步/自动循环运行中（总）
OR W289.00  ; RK_12 预焊上下料机构单步标志
ANDLD
OUT TR2
AND D1235.03  ; RK_12 预焊上下料机构下料Z轴OK|#1|#2NG放料位4（步）
AND 856.06  ; RK_12 U4_X 预焊上下料X轴OK放料位标志
AND W289.09  ; 出料拉带有放OK电池需求标志
AND H96.05  ; RK_12 预焊上下料机构下料夹爪有MES校验完成OK料记忆
ANDNOT H96.06  ; RK_12 预焊上下料机构下料夹爪有MES校验完成NG料记忆
ANDNOT 2054.13  ; RK_12 U4_Z 预焊下料Z轴忙标志位
ANDNOT W286.13  ; RK_12 U4_Z 预焊下料Z轴轴忙标志
OUT 558.03  ; RK_12 U4_Z 预焊下料Z轴OK放料位条件
TIMHX(551) 0683 D24  ; 伺服启动延时, RK_12 U4_Z 预焊下料Z轴OK放料位延时[A]
LD TR2
LD 558.03  ; RK_12 U4_Z 预焊下料Z轴OK放料位条件
AND T0683  ; RK_12 U4_Z 预焊下料Z轴OK放料位延时[A]
OR 658.03  ; RK_12 U4_Z 预焊下料Z轴OK放料位[A]
ANDLD
ANDNOT W287.08  ; RK_12 U4_Z 预焊下料Z轴OK放料位完成标志
OUT 658.03  ; RK_12 U4_Z 预焊下料Z轴OK放料位[A]
LD TR1
LD 458.03  ; RK_12 U4_Z 预焊下料Z轴OK放料位[M]
OR 658.03  ; RK_12 U4_Z 预焊下料Z轴OK放料位[A]
ANDLD
ANDNOT 2054.13  ; RK_12 U4_Z 预焊下料Z轴忙标志位
OUT 158.03  ; RK_12 U4_Z 预焊下料Z轴OK放料位触发
LD TR0
LD 458.03  ; RK_12 U4_Z 预焊下料Z轴OK放料位[M]
OR 658.03  ; RK_12 U4_Z 预焊下料Z轴OK放料位[A]
AND 2054.13  ; RK_12 U4_Z 预焊下料Z轴忙标志位
AND P_1s
OR 858.03  ; RK_12 U4_Z 预焊下料Z轴OK放料位标志
ANDLD
OUT 958.03  ; RK_12 U4_Z 预焊下料Z轴OK放料位[lamp]

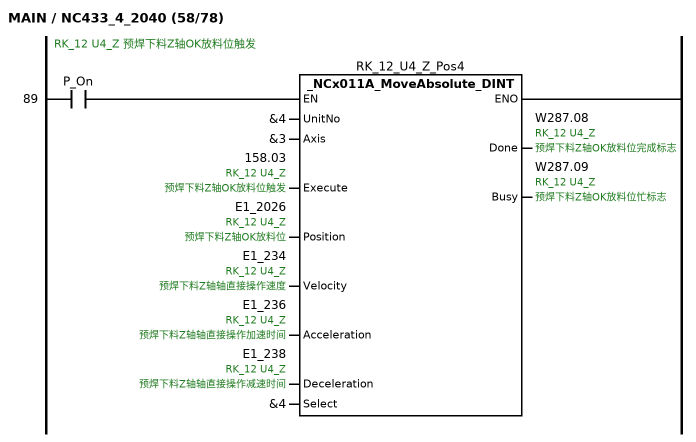
; rung 89: RK_12 U4_Z 预焊下料Z轴OK放料位触发
LD P_On
CALL RK_12_U4_Z_Pos4 : _NCx011A_MoveAbsolute_DINT (UnitNo := &4, Axis := &3, Execute := 158.03, Position := E1_2026, Velocity := E1_234, Acceleration := E1_236, Deceleration := E1_238, Select := &4, Done => W287.08, Busy => W287.09)  ; RK_12 U4_Z 预焊下料Z轴OK放料位触发, RK_12 U4_Z 预焊下料Z轴OK放料位, RK_12 U4_Z 预焊下料Z轴轴直接操作速度, RK_12 U4_Z 预焊下料Z轴轴直接操作加速时间, RK_12 U4_Z 预焊下料Z轴轴直接操作减速时间, RK_12 U4_Z 预焊下料Z轴OK放料位完成标志, RK_12 U4_Z 预焊下料Z轴OK放料位忙标志

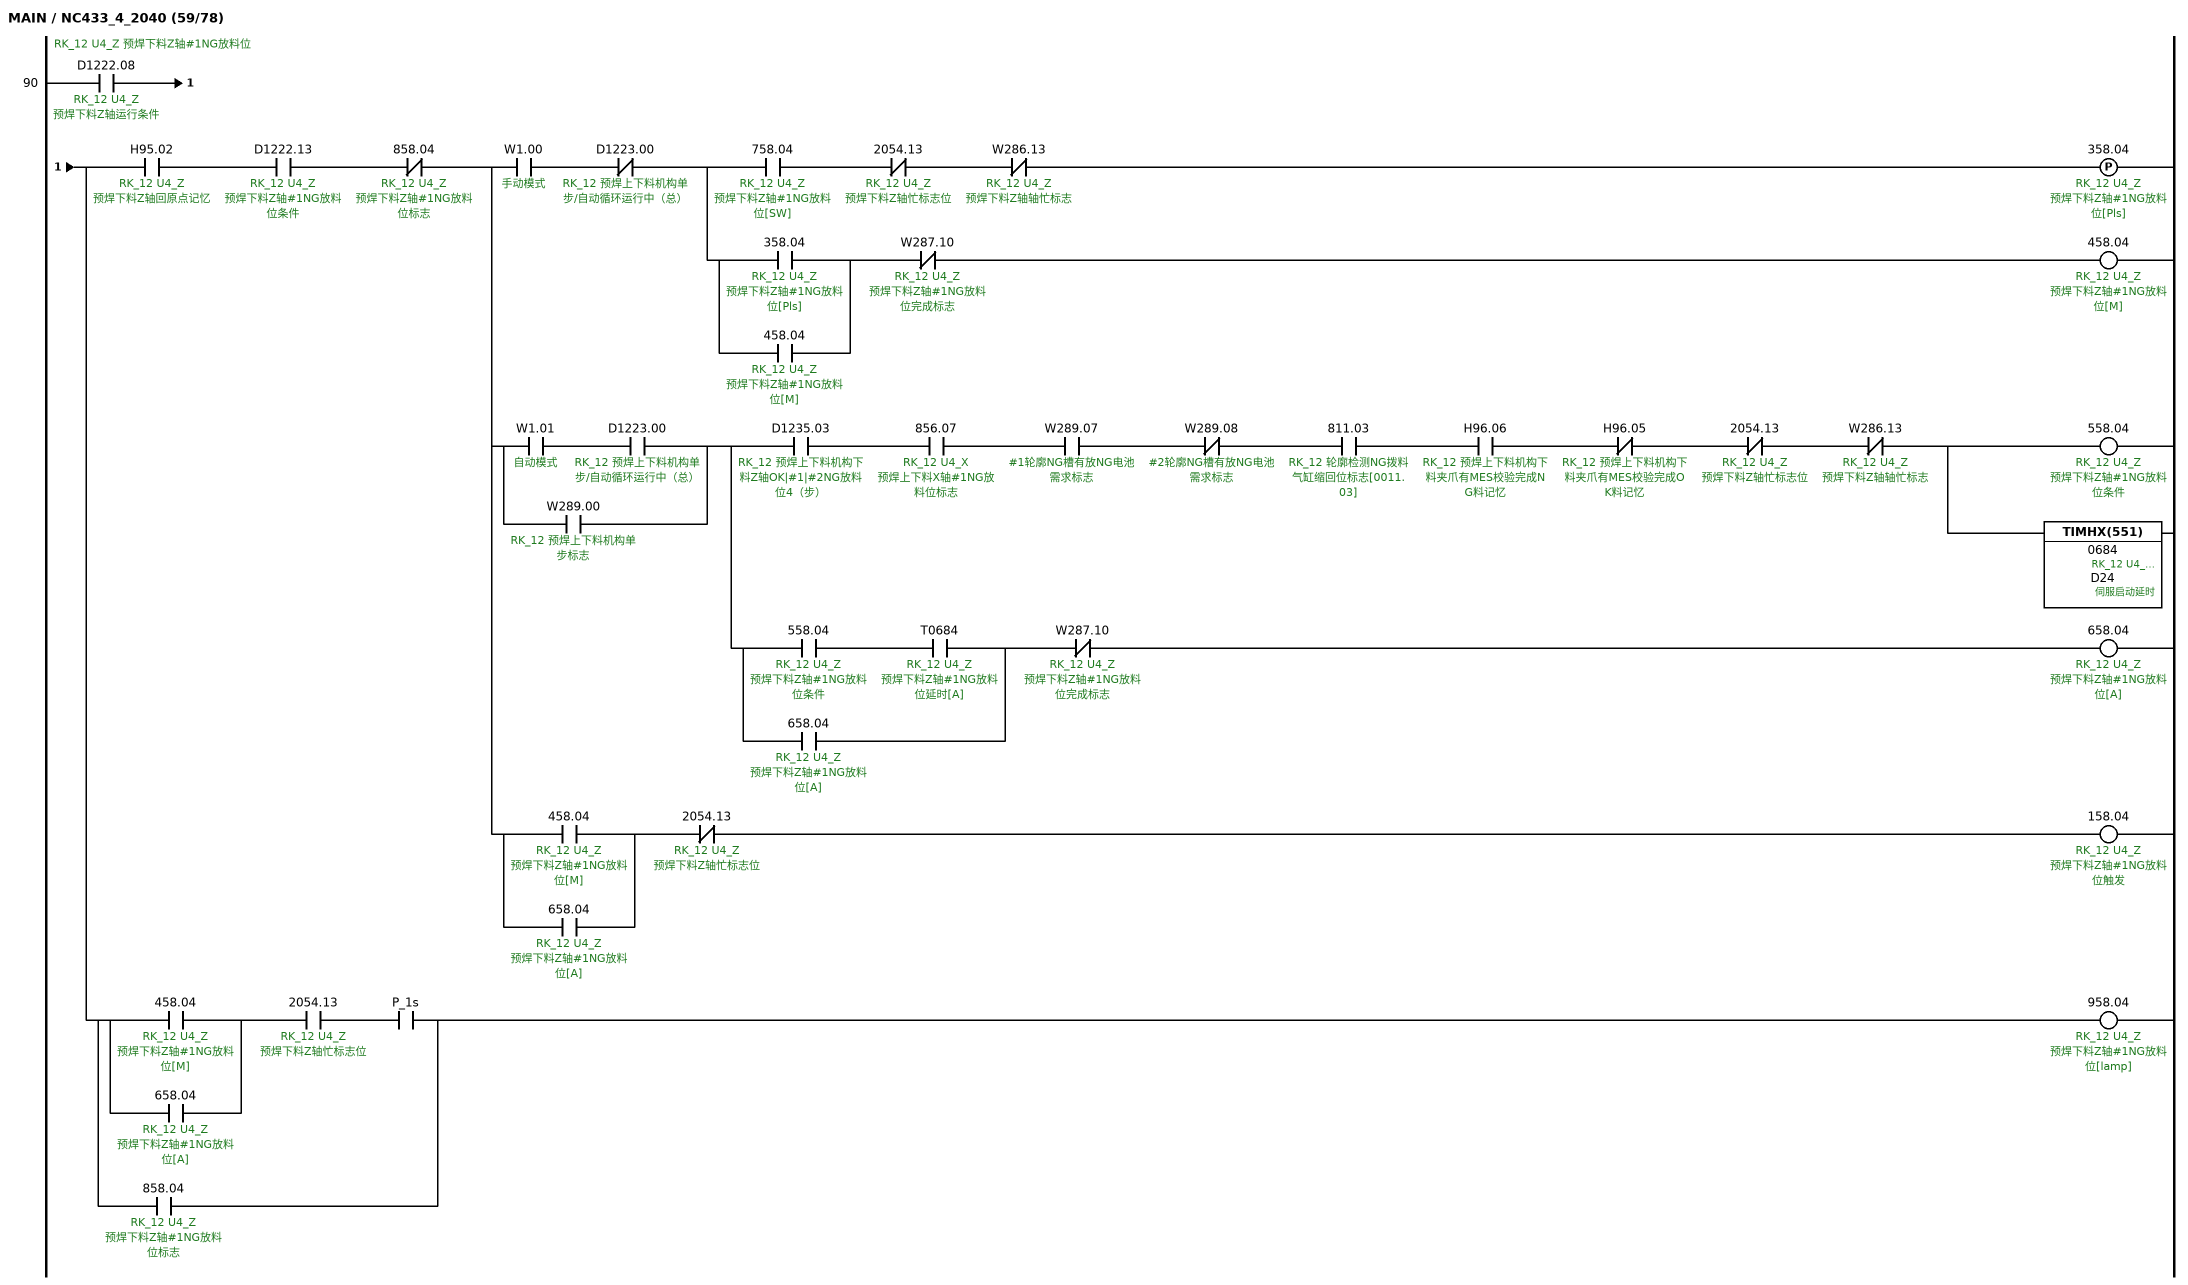
; rung 90: RK_12 U4_Z 预焊下料Z轴#1NG放料位
LD D1222.08  ; RK_12 U4_Z 预焊下料Z轴运行条件
OUT TR0
AND H95.02  ; RK_12 U4_Z 预焊下料Z轴回原点记忆
AND D1222.13  ; RK_12 U4_Z 预焊下料Z轴#1NG放料位条件
ANDNOT 858.04  ; RK_12 U4_Z 预焊下料Z轴#1NG放料位标志
OUT TR1
AND W1.00  ; 手动模式
ANDNOT D1223.00  ; RK_12 预焊上下料机构单步/自动循环运行中（总）
OUT TR2
AND 758.04  ; RK_12 U4_Z 预焊下料Z轴#1NG放料位[SW]
ANDNOT 2054.13  ; RK_12 U4_Z 预焊下料Z轴忙标志位
ANDNOT W286.13  ; RK_12 U4_Z 预焊下料Z轴轴忙标志
DIFU(013) 358.04  ; RK_12 U4_Z 预焊下料Z轴#1NG放料位[Pls]
LD TR2
LD 358.04  ; RK_12 U4_Z 预焊下料Z轴#1NG放料位[Pls]
OR 458.04  ; RK_12 U4_Z 预焊下料Z轴#1NG放料位[M]
ANDLD
ANDNOT W287.10  ; RK_12 U4_Z 预焊下料Z轴#1NG放料位完成标志
OUT 458.04  ; RK_12 U4_Z 预焊下料Z轴#1NG放料位[M]
LD TR1
LD W1.01  ; 自动模式
AND D1223.00  ; RK_12 预焊上下料机构单步/自动循环运行中（总）
OR W289.00  ; RK_12 预焊上下料机构单步标志
ANDLD
OUT TR2
AND D1235.03  ; RK_12 预焊上下料机构下料Z轴OK|#1|#2NG放料位4（步）
AND 856.07  ; RK_12 U4_X 预焊上下料X轴#1NG放料位标志
AND W289.07  ; #1轮廓NG槽有放NG电池需求标志
ANDNOT W289.08  ; #2轮廓NG槽有放NG电池需求标志
AND 811.03  ; RK_12 轮廓检测NG拨料气缸缩回位标志[0011.03]
AND H96.06  ; RK_12 预焊上下料机构下料夹爪有MES校验完成NG料记忆
ANDNOT H96.05  ; RK_12 预焊上下料机构下料夹爪有MES校验完成OK料记忆
ANDNOT 2054.13  ; RK_12 U4_Z 预焊下料Z轴忙标志位
ANDNOT W286.13  ; RK_12 U4_Z 预焊下料Z轴轴忙标志
OUT 558.04  ; RK_12 U4_Z 预焊下料Z轴#1NG放料位条件
TIMHX(551) 0684 D24  ; 伺服启动延时, RK_12 U4_Z 预焊下料Z轴#1NG放料位延时[A]
LD TR2
LD 558.04  ; RK_12 U4_Z 预焊下料Z轴#1NG放料位条件
AND T0684  ; RK_12 U4_Z 预焊下料Z轴#1NG放料位延时[A]
OR 658.04  ; RK_12 U4_Z 预焊下料Z轴#1NG放料位[A]
ANDLD
ANDNOT W287.10  ; RK_12 U4_Z 预焊下料Z轴#1NG放料位完成标志
OUT 658.04  ; RK_12 U4_Z 预焊下料Z轴#1NG放料位[A]
LD TR1
LD 458.04  ; RK_12 U4_Z 预焊下料Z轴#1NG放料位[M]
OR 658.04  ; RK_12 U4_Z 预焊下料Z轴#1NG放料位[A]
ANDLD
ANDNOT 2054.13  ; RK_12 U4_Z 预焊下料Z轴忙标志位
OUT 158.04  ; RK_12 U4_Z 预焊下料Z轴#1NG放料位触发
LD TR0
LD 458.04  ; RK_12 U4_Z 预焊下料Z轴#1NG放料位[M]
OR 658.04  ; RK_12 U4_Z 预焊下料Z轴#1NG放料位[A]
AND 2054.13  ; RK_12 U4_Z 预焊下料Z轴忙标志位
AND P_1s
OR 858.04  ; RK_12 U4_Z 预焊下料Z轴#1NG放料位标志
ANDLD
OUT 958.04  ; RK_12 U4_Z 预焊下料Z轴#1NG放料位[lamp]

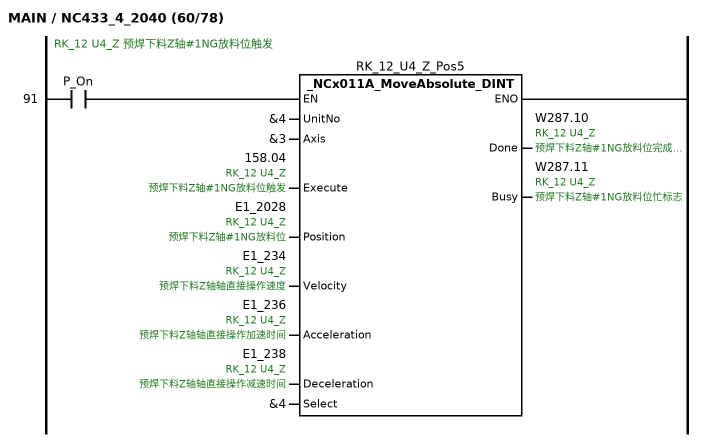
; rung 91: RK_12 U4_Z 预焊下料Z轴#1NG放料位触发
LD P_On
CALL RK_12_U4_Z_Pos5 : _NCx011A_MoveAbsolute_DINT (UnitNo := &4, Axis := &3, Execute := 158.04, Position := E1_2028, Velocity := E1_234, Acceleration := E1_236, Deceleration := E1_238, Select := &4, Done => W287.10, Busy => W287.11)  ; RK_12 U4_Z 预焊下料Z轴#1NG放料位触发, RK_12 U4_Z 预焊下料Z轴#1NG放料位, RK_12 U4_Z 预焊下料Z轴轴直接操作速度, RK_12 U4_Z 预焊下料Z轴轴直接操作加速时间, RK_12 U4_Z 预焊下料Z轴轴直接操作减速时间, RK_12 U4_Z 预焊下料Z轴#1NG放料位完成标志, RK_12 U4_Z 预焊下料Z轴#1NG放料位忙标志

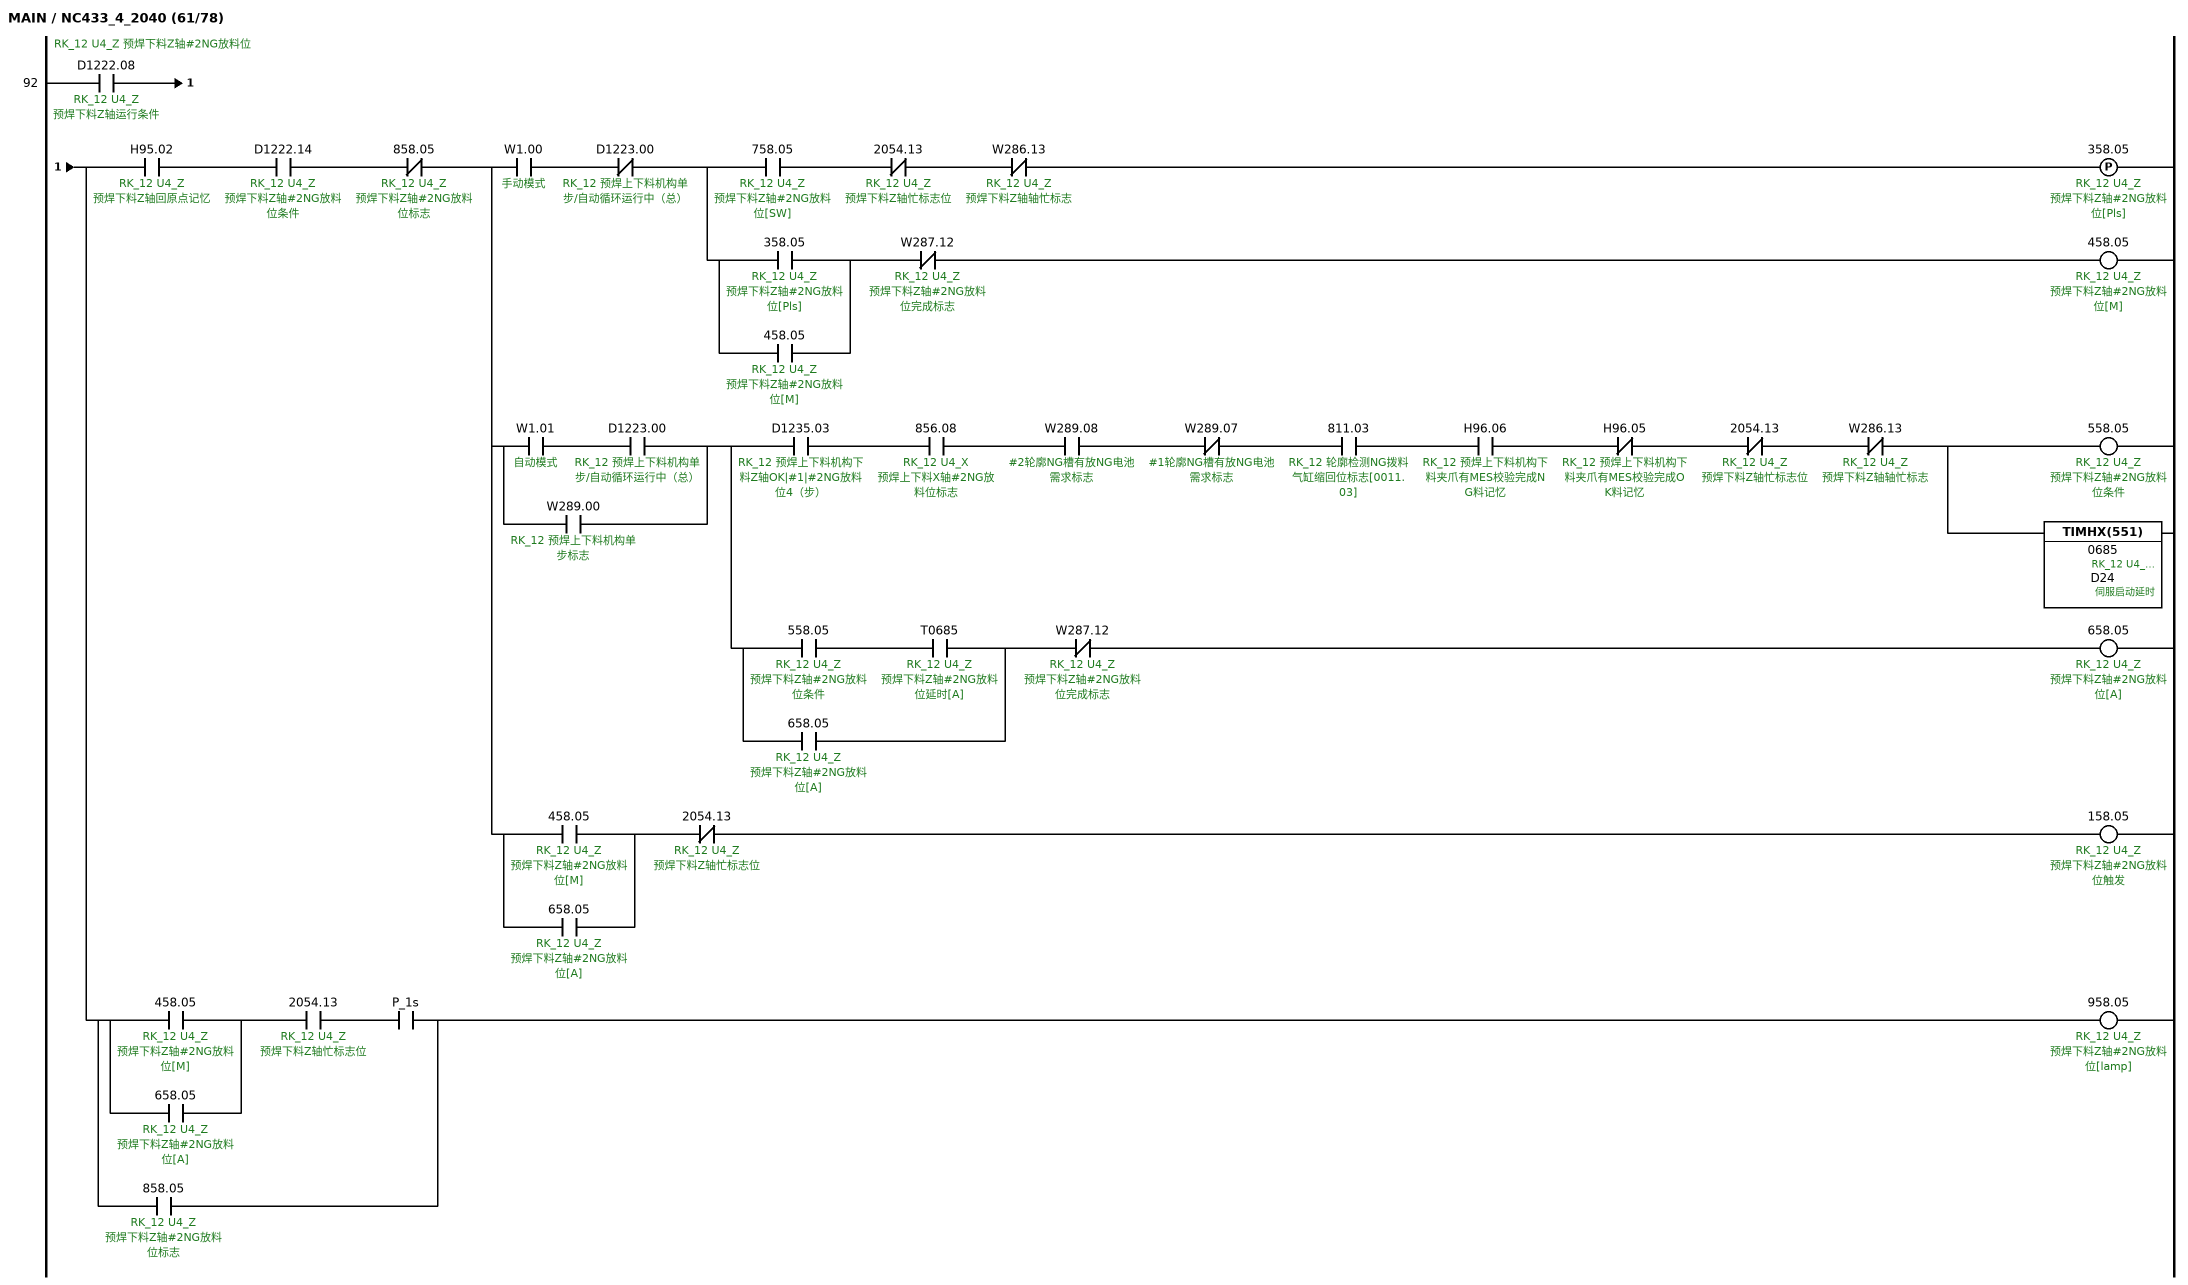
; rung 92: RK_12 U4_Z 预焊下料Z轴#2NG放料位
LD D1222.08  ; RK_12 U4_Z 预焊下料Z轴运行条件
OUT TR0
AND H95.02  ; RK_12 U4_Z 预焊下料Z轴回原点记忆
AND D1222.14  ; RK_12 U4_Z 预焊下料Z轴#2NG放料位条件
ANDNOT 858.05  ; RK_12 U4_Z 预焊下料Z轴#2NG放料位标志
OUT TR1
AND W1.00  ; 手动模式
ANDNOT D1223.00  ; RK_12 预焊上下料机构单步/自动循环运行中（总）
OUT TR2
AND 758.05  ; RK_12 U4_Z 预焊下料Z轴#2NG放料位[SW]
ANDNOT 2054.13  ; RK_12 U4_Z 预焊下料Z轴忙标志位
ANDNOT W286.13  ; RK_12 U4_Z 预焊下料Z轴轴忙标志
DIFU(013) 358.05  ; RK_12 U4_Z 预焊下料Z轴#2NG放料位[Pls]
LD TR2
LD 358.05  ; RK_12 U4_Z 预焊下料Z轴#2NG放料位[Pls]
OR 458.05  ; RK_12 U4_Z 预焊下料Z轴#2NG放料位[M]
ANDLD
ANDNOT W287.12  ; RK_12 U4_Z 预焊下料Z轴#2NG放料位完成标志
OUT 458.05  ; RK_12 U4_Z 预焊下料Z轴#2NG放料位[M]
LD TR1
LD W1.01  ; 自动模式
AND D1223.00  ; RK_12 预焊上下料机构单步/自动循环运行中（总）
OR W289.00  ; RK_12 预焊上下料机构单步标志
ANDLD
OUT TR2
AND D1235.03  ; RK_12 预焊上下料机构下料Z轴OK|#1|#2NG放料位4（步）
AND 856.08  ; RK_12 U4_X 预焊上下料X轴#2NG放料位标志
AND W289.08  ; #2轮廓NG槽有放NG电池需求标志
ANDNOT W289.07  ; #1轮廓NG槽有放NG电池需求标志
AND 811.03  ; RK_12 轮廓检测NG拨料气缸缩回位标志[0011.03]
AND H96.06  ; RK_12 预焊上下料机构下料夹爪有MES校验完成NG料记忆
ANDNOT H96.05  ; RK_12 预焊上下料机构下料夹爪有MES校验完成OK料记忆
ANDNOT 2054.13  ; RK_12 U4_Z 预焊下料Z轴忙标志位
ANDNOT W286.13  ; RK_12 U4_Z 预焊下料Z轴轴忙标志
OUT 558.05  ; RK_12 U4_Z 预焊下料Z轴#2NG放料位条件
TIMHX(551) 0685 D24  ; 伺服启动延时, RK_12 U4_Z 预焊下料Z轴#2NG放料位延时[A]
LD TR2
LD 558.05  ; RK_12 U4_Z 预焊下料Z轴#2NG放料位条件
AND T0685  ; RK_12 U4_Z 预焊下料Z轴#2NG放料位延时[A]
OR 658.05  ; RK_12 U4_Z 预焊下料Z轴#2NG放料位[A]
ANDLD
ANDNOT W287.12  ; RK_12 U4_Z 预焊下料Z轴#2NG放料位完成标志
OUT 658.05  ; RK_12 U4_Z 预焊下料Z轴#2NG放料位[A]
LD TR1
LD 458.05  ; RK_12 U4_Z 预焊下料Z轴#2NG放料位[M]
OR 658.05  ; RK_12 U4_Z 预焊下料Z轴#2NG放料位[A]
ANDLD
ANDNOT 2054.13  ; RK_12 U4_Z 预焊下料Z轴忙标志位
OUT 158.05  ; RK_12 U4_Z 预焊下料Z轴#2NG放料位触发
LD TR0
LD 458.05  ; RK_12 U4_Z 预焊下料Z轴#2NG放料位[M]
OR 658.05  ; RK_12 U4_Z 预焊下料Z轴#2NG放料位[A]
AND 2054.13  ; RK_12 U4_Z 预焊下料Z轴忙标志位
AND P_1s
OR 858.05  ; RK_12 U4_Z 预焊下料Z轴#2NG放料位标志
ANDLD
OUT 958.05  ; RK_12 U4_Z 预焊下料Z轴#2NG放料位[lamp]

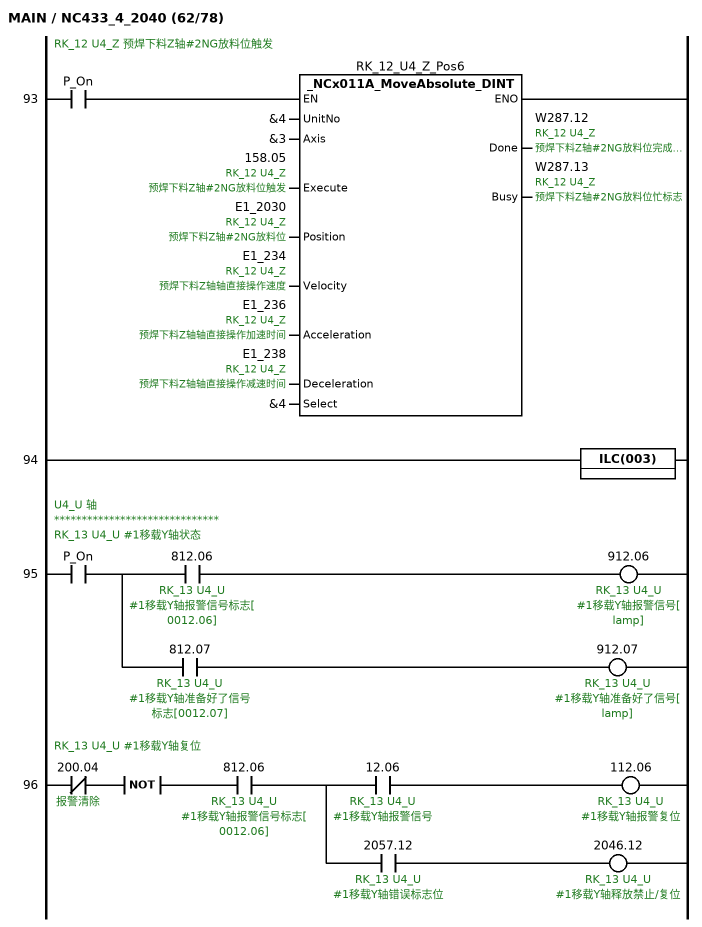
; rung 93: RK_12 U4_Z 预焊下料Z轴#2NG放料位触发
LD P_On
CALL RK_12_U4_Z_Pos6 : _NCx011A_MoveAbsolute_DINT (UnitNo := &4, Axis := &3, Execute := 158.05, Position := E1_2030, Velocity := E1_234, Acceleration := E1_236, Deceleration := E1_238, Select := &4, Done => W287.12, Busy => W287.13)  ; RK_12 U4_Z 预焊下料Z轴#2NG放料位触发, RK_12 U4_Z 预焊下料Z轴#2NG放料位, RK_12 U4_Z 预焊下料Z轴轴直接操作速度, RK_12 U4_Z 预焊下料Z轴轴直接操作加速时间, RK_12 U4_Z 预焊下料Z轴轴直接操作减速时间, RK_12 U4_Z 预焊下料Z轴#2NG放料位完成标志, RK_12 U4_Z 预焊下料Z轴#2NG放料位忙标志
; rung 94
ILC(003)
; rung 95: U4_U 轴 / ****************************** / RK_13 U4_U #1移载Y轴状态
LD P_On
OUT TR0
AND 812.06  ; RK_13 U4_U #1移载Y轴报警信号标志[0012.06]
OUT 912.06  ; RK_13 U4_U #1移载Y轴报警信号[lamp]
LD TR0
AND 812.07  ; RK_13 U4_U #1移载Y轴准备好了信号标志[0012.07]
OUT 912.07  ; RK_13 U4_U #1移载Y轴准备好了信号[lamp]
; rung 96: RK_13 U4_U #1移载Y轴复位
LDNOT 200.04  ; 报警清除
NOT(520)
AND 812.06  ; RK_13 U4_U #1移载Y轴报警信号标志[0012.06]
OUT TR0
AND 12.06  ; RK_13 U4_U #1移载Y轴报警信号
OUT 112.06  ; RK_13 U4_U #1移载Y轴报警复位
LD TR0
AND 2057.12  ; RK_13 U4_U #1移载Y轴错误标志位
OUT 2046.12  ; RK_13 U4_U #1移载Y轴释放禁止/复位

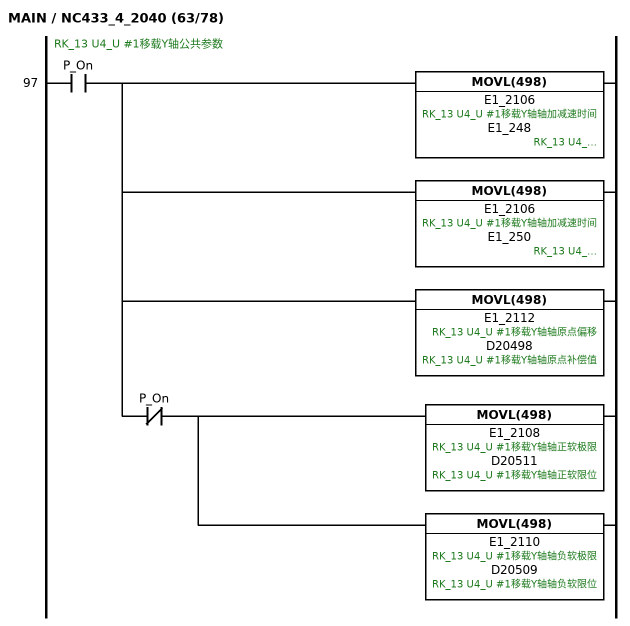
; rung 97: RK_13 U4_U #1移载Y轴公共参数
LD P_On
MOVL(498) E1_2106 E1_248  ; RK_13 U4_U #1移载Y轴轴加减速时间, RK_13 U4_U #1移载Y轴轴直接操作加速时间
MOVL(498) E1_2106 E1_250  ; RK_13 U4_U #1移载Y轴轴加减速时间, RK_13 U4_U #1移载Y轴轴直接操作减速时间
MOVL(498) E1_2112 D20498  ; RK_13 U4_U #1移载Y轴轴原点偏移, RK_13 U4_U #1移载Y轴轴原点补偿值
ANDNOT P_On
MOVL(498) E1_2108 D20511  ; RK_13 U4_U #1移载Y轴轴正软极限, RK_13 U4_U #1移载Y轴轴正软限位
MOVL(498) E1_2110 D20509  ; RK_13 U4_U #1移载Y轴轴负软极限, RK_13 U4_U #1移载Y轴轴负软限位

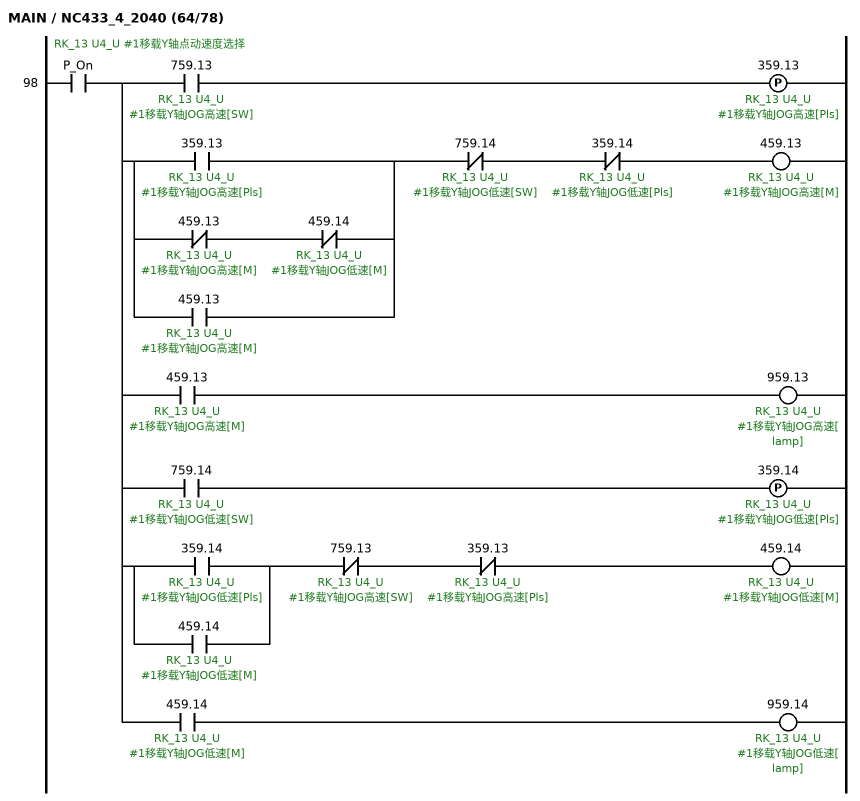
; rung 98: RK_13 U4_U #1移载Y轴点动速度选择
LD P_On
OUT TR0
AND 759.13  ; RK_13 U4_U #1移载Y轴JOG高速[SW]
DIFU(013) 359.13  ; RK_13 U4_U #1移载Y轴JOG高速[Pls]
LD TR0
LD 359.13  ; RK_13 U4_U #1移载Y轴JOG高速[Pls]
LDNOT 459.13  ; RK_13 U4_U #1移载Y轴JOG高速[M]
ANDNOT 459.14  ; RK_13 U4_U #1移载Y轴JOG低速[M]
ORLD
OR 459.13  ; RK_13 U4_U #1移载Y轴JOG高速[M]
ANDLD
ANDNOT 759.14  ; RK_13 U4_U #1移载Y轴JOG低速[SW]
ANDNOT 359.14  ; RK_13 U4_U #1移载Y轴JOG低速[Pls]
OUT 459.13  ; RK_13 U4_U #1移载Y轴JOG高速[M]
LD TR0
AND 459.13  ; RK_13 U4_U #1移载Y轴JOG高速[M]
OUT 959.13  ; RK_13 U4_U #1移载Y轴JOG高速[lamp]
LD TR0
AND 759.14  ; RK_13 U4_U #1移载Y轴JOG低速[SW]
DIFU(013) 359.14  ; RK_13 U4_U #1移载Y轴JOG低速[Pls]
LD TR0
LD 359.14  ; RK_13 U4_U #1移载Y轴JOG低速[Pls]
OR 459.14  ; RK_13 U4_U #1移载Y轴JOG低速[M]
ANDLD
ANDNOT 759.13  ; RK_13 U4_U #1移载Y轴JOG高速[SW]
ANDNOT 359.13  ; RK_13 U4_U #1移载Y轴JOG高速[Pls]
OUT 459.14  ; RK_13 U4_U #1移载Y轴JOG低速[M]
LD TR0
AND 459.14  ; RK_13 U4_U #1移载Y轴JOG低速[M]
OUT 959.14  ; RK_13 U4_U #1移载Y轴JOG低速[lamp]

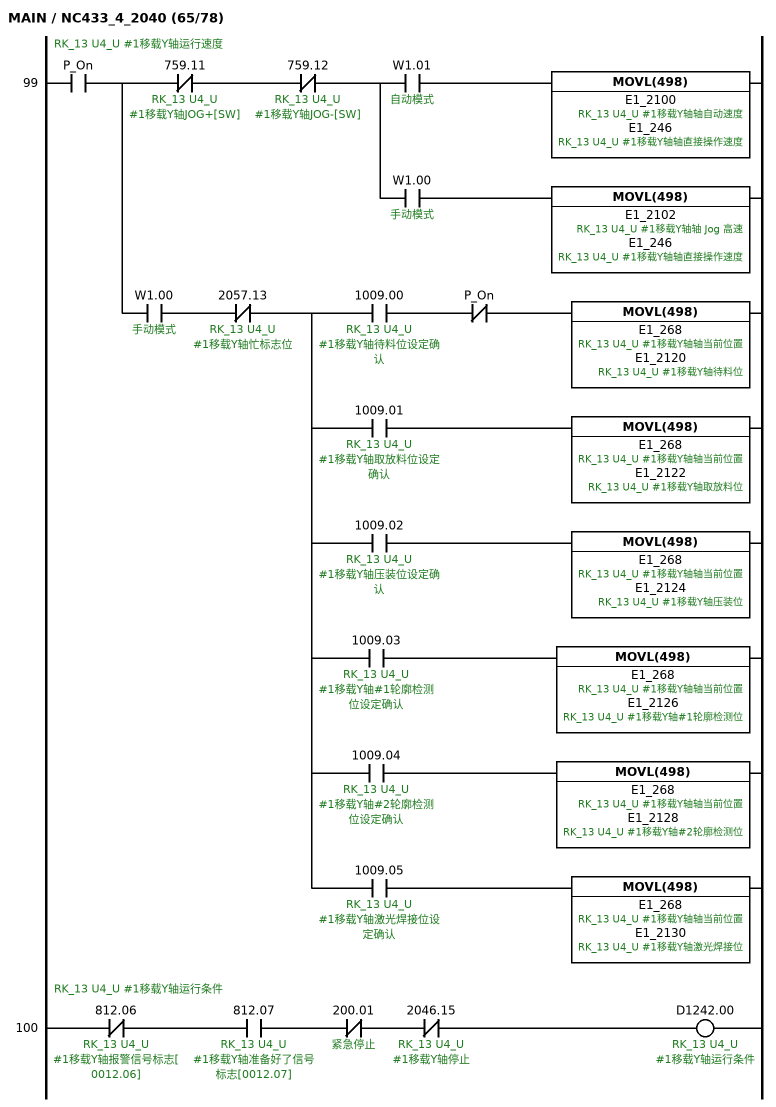
; rung 99: RK_13 U4_U #1移载Y轴运行速度
LD P_On
OUT TR0
ANDNOT 759.11  ; RK_13 U4_U #1移载Y轴JOG+[SW]
ANDNOT 759.12  ; RK_13 U4_U #1移载Y轴JOG-[SW]
OUT TR1
AND W1.01  ; 自动模式
MOVL(498) E1_2100 E1_246  ; RK_13 U4_U #1移载Y轴轴自动速度, RK_13 U4_U #1移载Y轴轴直接操作速度
LD TR1
AND W1.00  ; 手动模式
MOVL(498) E1_2102 E1_246  ; RK_13 U4_U #1移载Y轴轴 Jog 高速, RK_13 U4_U #1移载Y轴轴直接操作速度
LD TR0
AND W1.00  ; 手动模式
ANDNOT 2057.13  ; RK_13 U4_U #1移载Y轴忙标志位
OUT TR0
AND 1009.00  ; RK_13 U4_U #1移载Y轴待料位设定确认
ANDNOT P_On
MOVL(498) E1_268 E1_2120  ; RK_13 U4_U #1移载Y轴轴当前位置, RK_13 U4_U #1移载Y轴待料位
LD TR0
AND 1009.01  ; RK_13 U4_U #1移载Y轴取放料位设定确认
MOVL(498) E1_268 E1_2122  ; RK_13 U4_U #1移载Y轴轴当前位置, RK_13 U4_U #1移载Y轴取放料位
LD TR0
AND 1009.02  ; RK_13 U4_U #1移载Y轴压装位设定确认
MOVL(498) E1_268 E1_2124  ; RK_13 U4_U #1移载Y轴轴当前位置, RK_13 U4_U #1移载Y轴压装位
LD TR0
AND 1009.03  ; RK_13 U4_U #1移载Y轴#1轮廓检测位设定确认
MOVL(498) E1_268 E1_2126  ; RK_13 U4_U #1移载Y轴轴当前位置, RK_13 U4_U #1移载Y轴#1轮廓检测位
LD TR0
AND 1009.04  ; RK_13 U4_U #1移载Y轴#2轮廓检测位设定确认
MOVL(498) E1_268 E1_2128  ; RK_13 U4_U #1移载Y轴轴当前位置, RK_13 U4_U #1移载Y轴#2轮廓检测位
LD TR0
AND 1009.05  ; RK_13 U4_U #1移载Y轴激光焊接位设定确认
MOVL(498) E1_268 E1_2130  ; RK_13 U4_U #1移载Y轴轴当前位置, RK_13 U4_U #1移载Y轴激光焊接位
; rung 100: RK_13 U4_U #1移载Y轴运行条件
LDNOT 812.06  ; RK_13 U4_U #1移载Y轴报警信号标志[0012.06]
AND 812.07  ; RK_13 U4_U #1移载Y轴准备好了信号标志[0012.07]
ANDNOT 200.01  ; 紧急停止
ANDNOT 2046.15  ; RK_13 U4_U #1移载Y轴停止
OUT D1242.00  ; RK_13 U4_U #1移载Y轴运行条件

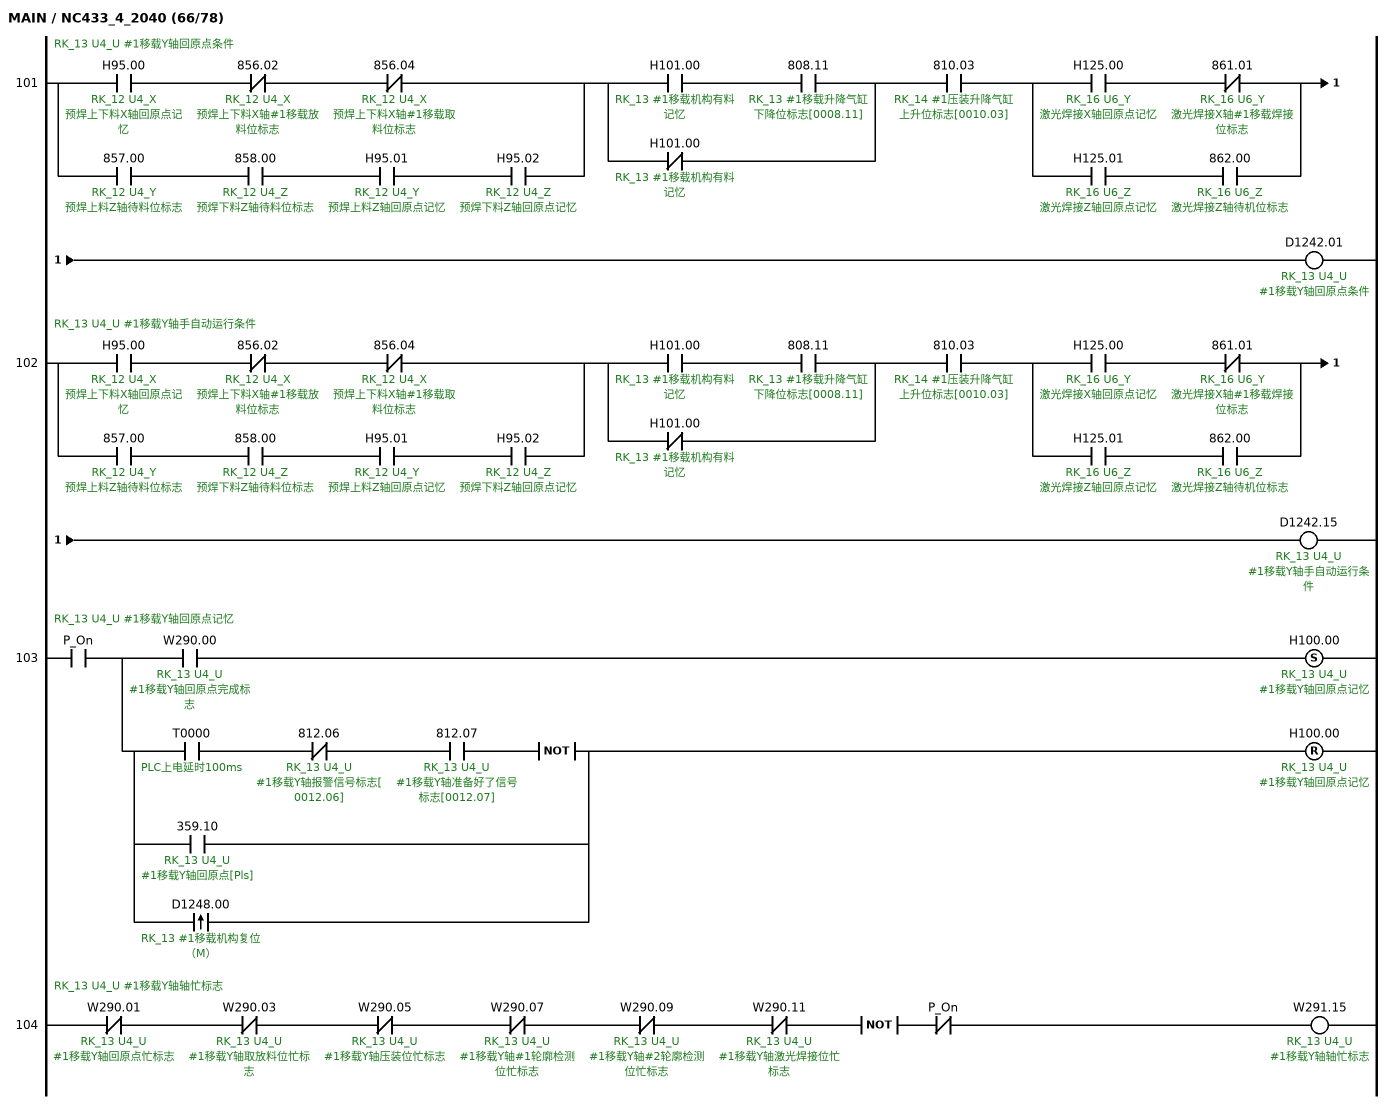
; rung 101: RK_13 U4_U #1移载Y轴回原点条件
LD H95.00  ; RK_12 U4_X 预焊上下料X轴回原点记忆
ANDNOT 856.02  ; RK_12 U4_X 预焊上下料X轴#1移载放料位标志
ANDNOT 856.04  ; RK_12 U4_X 预焊上下料X轴#1移载取料位标志
LD 857.00  ; RK_12 U4_Y 预焊上料Z轴待料位标志
AND 858.00  ; RK_12 U4_Z 预焊下料Z轴待料位标志
AND H95.01  ; RK_12 U4_Y 预焊上料Z轴回原点记忆
AND H95.02  ; RK_12 U4_Z 预焊下料Z轴回原点记忆
ORLD
LD H101.00  ; RK_13 #1移载机构有料记忆
AND 808.11  ; RK_13 #1移载升降气缸下降位标志[0008.11]
ORNOT H101.00  ; RK_13 #1移载机构有料记忆
ANDLD
AND 810.03  ; RK_14 #1压装升降气缸上升位标志[0010.03]
LD H125.00  ; RK_16 U6_Y 激光焊接X轴回原点记忆
ANDNOT 861.01  ; RK_16 U6_Y 激光焊接X轴#1移载焊接位标志
LD H125.01  ; RK_16 U6_Z 激光焊接Z轴回原点记忆
AND 862.00  ; RK_16 U6_Z 激光焊接Z轴待机位标志
ORLD
ANDLD
OUT D1242.01  ; RK_13 U4_U #1移载Y轴回原点条件
; rung 102: RK_13 U4_U #1移载Y轴手自动运行条件
LD H95.00  ; RK_12 U4_X 预焊上下料X轴回原点记忆
ANDNOT 856.02  ; RK_12 U4_X 预焊上下料X轴#1移载放料位标志
ANDNOT 856.04  ; RK_12 U4_X 预焊上下料X轴#1移载取料位标志
LD 857.00  ; RK_12 U4_Y 预焊上料Z轴待料位标志
AND 858.00  ; RK_12 U4_Z 预焊下料Z轴待料位标志
AND H95.01  ; RK_12 U4_Y 预焊上料Z轴回原点记忆
AND H95.02  ; RK_12 U4_Z 预焊下料Z轴回原点记忆
ORLD
LD H101.00  ; RK_13 #1移载机构有料记忆
AND 808.11  ; RK_13 #1移载升降气缸下降位标志[0008.11]
ORNOT H101.00  ; RK_13 #1移载机构有料记忆
ANDLD
AND 810.03  ; RK_14 #1压装升降气缸上升位标志[0010.03]
LD H125.00  ; RK_16 U6_Y 激光焊接X轴回原点记忆
ANDNOT 861.01  ; RK_16 U6_Y 激光焊接X轴#1移载焊接位标志
LD H125.01  ; RK_16 U6_Z 激光焊接Z轴回原点记忆
AND 862.00  ; RK_16 U6_Z 激光焊接Z轴待机位标志
ORLD
ANDLD
OUT D1242.15  ; RK_13 U4_U #1移载Y轴手自动运行条件
; rung 103: RK_13 U4_U #1移载Y轴回原点记忆
LD P_On
OUT TR0
AND W290.00  ; RK_13 U4_U #1移载Y轴回原点完成标志
SET H100.00  ; RK_13 U4_U #1移载Y轴回原点记忆
LD TR0
LD T0000  ; PLC上电延时100ms
ANDNOT 812.06  ; RK_13 U4_U #1移载Y轴报警信号标志[0012.06]
AND 812.07  ; RK_13 U4_U #1移载Y轴准备好了信号标志[0012.07]
NOT(520)
OR 359.10  ; RK_13 U4_U #1移载Y轴回原点[Pls]
@OR D1248.00  ; RK_13 #1移载机构复位（M）
ANDLD
RSET H100.00  ; RK_13 U4_U #1移载Y轴回原点记忆
; rung 104: RK_13 U4_U #1移载Y轴轴忙标志
LDNOT W290.01  ; RK_13 U4_U #1移载Y轴回原点忙标志
ANDNOT W290.03  ; RK_13 U4_U #1移载Y轴取放料位忙标志
ANDNOT W290.05  ; RK_13 U4_U #1移载Y轴压装位忙标志
ANDNOT W290.07  ; RK_13 U4_U #1移载Y轴#1轮廓检测位忙标志
ANDNOT W290.09  ; RK_13 U4_U #1移载Y轴#2轮廓检测位忙标志
ANDNOT W290.11  ; RK_13 U4_U #1移载Y轴激光焊接位忙标志
NOT(520)
ANDNOT P_On
OUT W291.15  ; RK_13 U4_U #1移载Y轴轴忙标志

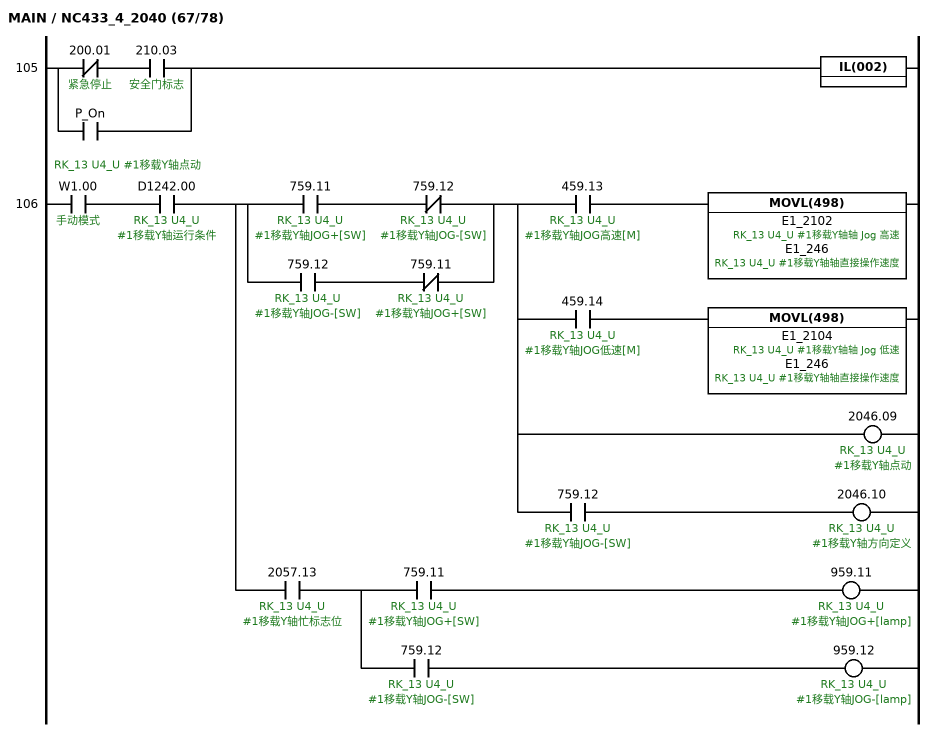
; rung 105
LDNOT 200.01  ; 紧急停止
AND 210.03  ; 安全门标志
OR P_On
IL(002)
; rung 106: RK_13 U4_U #1移载Y轴点动
LD W1.00  ; 手动模式
AND D1242.00  ; RK_13 U4_U #1移载Y轴运行条件
OUT TR0
LD 759.11  ; RK_13 U4_U #1移载Y轴JOG+[SW]
ANDNOT 759.12  ; RK_13 U4_U #1移载Y轴JOG-[SW]
LD 759.12  ; RK_13 U4_U #1移载Y轴JOG-[SW]
ANDNOT 759.11  ; RK_13 U4_U #1移载Y轴JOG+[SW]
ORLD
ANDLD
OUT TR1
AND 459.13  ; RK_13 U4_U #1移载Y轴JOG高速[M]
MOVL(498) E1_2102 E1_246  ; RK_13 U4_U #1移载Y轴轴 Jog 高速, RK_13 U4_U #1移载Y轴轴直接操作速度
LD TR1
AND 459.14  ; RK_13 U4_U #1移载Y轴JOG低速[M]
MOVL(498) E1_2104 E1_246  ; RK_13 U4_U #1移载Y轴轴 Jog 低速, RK_13 U4_U #1移载Y轴轴直接操作速度
LD TR1
OUT 2046.09  ; RK_13 U4_U #1移载Y轴点动
AND 759.12  ; RK_13 U4_U #1移载Y轴JOG-[SW]
OUT 2046.10  ; RK_13 U4_U #1移载Y轴方向定义
LD TR0
AND 2057.13  ; RK_13 U4_U #1移载Y轴忙标志位
OUT TR0
AND 759.11  ; RK_13 U4_U #1移载Y轴JOG+[SW]
OUT 959.11  ; RK_13 U4_U #1移载Y轴JOG+[lamp]
LD TR0
AND 759.12  ; RK_13 U4_U #1移载Y轴JOG-[SW]
OUT 959.12  ; RK_13 U4_U #1移载Y轴JOG-[lamp]

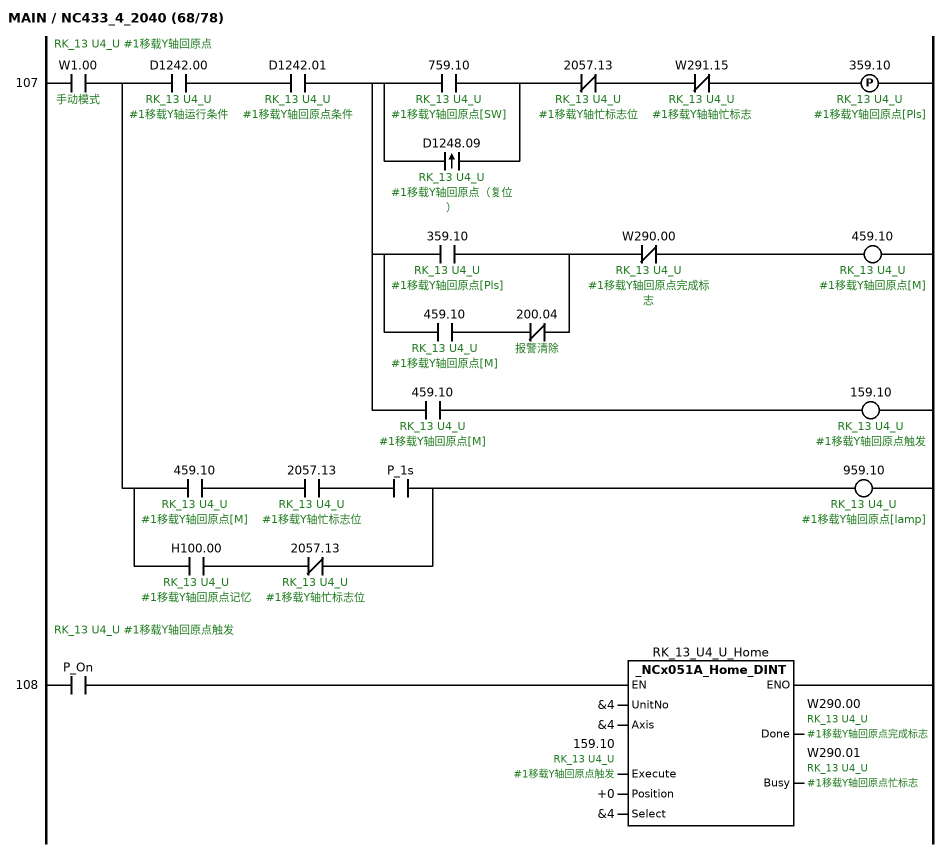
; rung 107: RK_13 U4_U #1移载Y轴回原点
LD W1.00  ; 手动模式
OUT TR0
AND D1242.00  ; RK_13 U4_U #1移载Y轴运行条件
AND D1242.01  ; RK_13 U4_U #1移载Y轴回原点条件
OUT TR1
LD 759.10  ; RK_13 U4_U #1移载Y轴回原点[SW]
@OR D1248.09  ; RK_13 U4_U #1移载Y轴回原点（复位）
ANDLD
ANDNOT 2057.13  ; RK_13 U4_U #1移载Y轴忙标志位
ANDNOT W291.15  ; RK_13 U4_U #1移载Y轴轴忙标志
DIFU(013) 359.10  ; RK_13 U4_U #1移载Y轴回原点[Pls]
LD TR1
LD 359.10  ; RK_13 U4_U #1移载Y轴回原点[Pls]
LD 459.10  ; RK_13 U4_U #1移载Y轴回原点[M]
ANDNOT 200.04  ; 报警清除
ORLD
ANDLD
ANDNOT W290.00  ; RK_13 U4_U #1移载Y轴回原点完成标志
OUT 459.10  ; RK_13 U4_U #1移载Y轴回原点[M]
LD TR1
AND 459.10  ; RK_13 U4_U #1移载Y轴回原点[M]
OUT 159.10  ; RK_13 U4_U #1移载Y轴回原点触发
LD TR0
LD 459.10  ; RK_13 U4_U #1移载Y轴回原点[M]
AND 2057.13  ; RK_13 U4_U #1移载Y轴忙标志位
AND P_1s
LD H100.00  ; RK_13 U4_U #1移载Y轴回原点记忆
ANDNOT 2057.13  ; RK_13 U4_U #1移载Y轴忙标志位
ORLD
ANDLD
OUT 959.10  ; RK_13 U4_U #1移载Y轴回原点[lamp]
; rung 108: RK_13 U4_U #1移载Y轴回原点触发
LD P_On
CALL RK_13_U4_U_Home : _NCx051A_Home_DINT (UnitNo := &4, Axis := &4, Execute := 159.10, Position := +0, Select := &4, Done => W290.00, Busy => W290.01)  ; RK_13 U4_U #1移载Y轴回原点触发, RK_13 U4_U #1移载Y轴回原点完成标志, RK_13 U4_U #1移载Y轴回原点忙标志

